// TwinCAT 3 PLC project Untitled1
// ProgramVersion: 3.1.4023.0
// libraries:
//   CmpBitmapPool, * (System)
//   Tc2_ControllerToolbox, * (Beckhoff Automation GmbH)
//   Tc2_Drive, * (Beckhoff Automation GmbH)
//   Tc2_EtherCAT, * (Beckhoff Automation GmbH)
//   Tc2_MC2, * (Beckhoff Automation GmbH)
//   Tc2_MC2_Camming, * (Beckhoff Automation GmbH)
//   Tc2_MC2_Drive, * (Beckhoff Automation GmbH)
//   Tc2_MC2_FlyingSaw, * (Beckhoff Automation GmbH)
//   Tc2_Standard, * (Beckhoff Automation GmbH)
//   Tc2_System, * (Beckhoff Automation GmbH)
//   Tc2_TcpIp, * (Beckhoff Automation GmbH)
//   Tc2_Utilities, * (Beckhoff Automation GmbH)
//   Tc3_Module, * (Beckhoff Automation GmbH)
//   VisuDialogs, * (System)
//   Visu Utils, * (System)
//   VisuSymbols,3.5.10.0,System
// project tree:
//   DUTs/Ctrl/ Cmd_Typ.TcDUT, Ctrl_Typ.TcDUT, InverterCtrl_Typ.TcDUT, Parameters_Typ.TcDUT, Persistent_Typ.TcDUT, Status_Typ.TcDUT, UnwindCmd_Typ.TcDUT, UnwinderParameters_Typ.TcDUT
//   DUTs/IO/Encoder/ Encoder_Control_Typ.TcDUT, Encoder_Status_Typ.TcDUT, Encoder_Typ.TcDUT
//   DUTs/IO/ IO_In_Typ.TcDUT, IO_Out_Typ.TcDUT, IO_Typ.TcDUT, ST_BasicInverter.TcDUT, ST_InfoData.TcDUT, ST_WcState.TcDUT
//   DUTs/Motion/Axis Typ/Basic Typ/ Basic_axis_typ.TcDUT
//   DUTs/Motion/Axis Typ/Basic Typ/enumTyp/ eBasicAxisState.TcDUT, eDriveModeOfOperation.TcDUT, eHomeModeOption.TcDUT, enumDriveType.TcDUT, enumMotionObject.TcDUT, enum_DriveUpdateError.TcDUT, enum_DriveUpdateStatus.TcDUT, E_EncoderType.TcDUT
//   DUTs/Motion/Axis Typ/Basic Typ/Input/ Basic_Input_typ.TcDUT
//   DUTs/Motion/Axis Typ/Basic Typ/Input/Cmd/ Basic_Command_axis_typ.TcDUT
//   DUTs/Motion/Axis Typ/Basic Typ/Input/Params/ Bacis_Parameter_axis_typ.TcDUT, Drive_Parameter_typ.TcDUT, Motion_Limit_Parameter.TcDUT, ST_BasicHomeParam.TcDUT, ST_HomeAbsEncoder.TcDUT, ST_HomeAbsSwitch.TcDUT, ST_HomeLagErr.TcDUT, ST_HomeOptions.TcDUT
//   DUTs/Motion/Axis Typ/Basic Typ/Output/ Basic_Error_axis_typ.TcDUT, Basic_Output_typ.TcDUT
//   DUTs/Motion/Axis Typ/Basic Typ/Output/Monitor/ Basic_Monitor_axis_typ.TcDUT, Basic_Monitor_FileUpdate_axis_typ.TcDUT
//   DUTs/Motion/Axis Typ/Basic Typ/Output/Status/ Basic_MC_MoveVelocity_Status_typ.TcDUT, Basic_MC_Power_Status_typ.TcDUT, Basic_MC_Reset_Status_typ.TcDUT, Basic_MC_SetOverride_typ.TcDUT, Basic_Status_axis_typ.TcDUT, Basic_Status_typ.TcDUT, Drive_Status_typ.TcDUT, ReadStatus_typ.TcDUT
//   DUTs/Motion/Axis Typ/CyclicAxis_Typ/ CyclicAxis_CMD_typ.TcDUT, CyclicAxis_Error_typ.TcDUT, CyclicAxis_Input_typ.TcDUT, CyclicAxis_monitor_typ.TcDUT, CyclicAxis_Output_typ.TcDUT, CyclicAxis_Param_typ.TcDUT, CyclicAxis_Status_typ.TcDUT, CyclicAxis_typ.TcDUT, CyclicPos_CMD_typ.TcDUT, CyclicPos_Param_typ.TcDUT, CyclicPos_Status_typ.TcDUT, CyclicVel_CMD_typ.TcDUT, CyclicVel_Param_typ.TcDUT, CyclicVel_Status_typ.TcDUT, eCyclicAxisState.TcDUT
//   DUTs/Motion/Axis Typ/ ExtendedAxisTyp_1.TcDUT, stAxisIF.TcDUT
//   DUTs/Motion/Axis Typ/MultiAxis_Typ/ CamIn_CMD_typ.TcDUT, CamIn_Param_typ.TcDUT, CamIn_Statuses_typ.TcDUT, CamOut_Param_typ.TcDUT, CamOut_Statuses_typ.TcDUT, CamTableSelectCMD_typ.TcDUT, CamTableSelect_Param_typ.TcDUT, CamTableSelect_Status_typ.TcDUT, eMultiAxisState.TcDUT, GearInDyn_CMD_typ.TcDUT, GearInDyn_Param_typ.TcDUT, GearInDyn_Statuses_typ.TcDUT, GearInMultiMaster_CMD_typ.TcDUT, GearInMultiMaster_Param_typ.TcDUT, GearInMultiMaster_Statuses_typ.TcDUT, GearInPos_CMD_typ.TcDUT, GearInPos_Param_typ.TcDUT, GearInPos_Statuses_typ.TcDUT, GearOut_Param_typ.TcDUT, GearOut_Statuses_typ.TcDUT, MultiAxis_CMD_typ.TcDUT, MultiAxis_Error_typ.TcDUT, MultiAxis_Input_typ.TcDUT, MultiAxis_monitor_typ.TcDUT, MultiAxis_Output_typ.TcDUT, MultiAxis_Param_typ.TcDUT, MultiAxis_Statuses_typ.TcDUT, MultiAxis_Status_typ.TcDUT, MultiAxis_typ.TcDUT
//   DUTs/Motion/Axis Typ/ParIDAccess_Typ/ eParIDAccessState.TcDUT, ParIDAccess_CMD_typ.TcDUT, ParIDAccess_Error_typ.TcDUT, ParIDAccess_Input_typ.TcDUT, ParIDAccess_monitor_typ.TcDUT, ParIDAccess_Output_typ.TcDUT, ParIDAccess_Param_typ.TcDUT, ParIDAccess_Par_ReadCoedSdo_typ.TcDUT, ParIDAccess_Par_WriteCoedSdo_typ.TcDUT, ParIDAccess_Status_axis_typ.TcDUT, ParIDAccess_Status_typ.TcDUT, ParIDAccess_Typ.TcDUT
//   DUTs/Motion/Axis Typ/VelocityCtrl/ eTorqueMode.TcDUT, eVelocityCtrlState.TcDUT, VelocityCtrl_CMD_typ.TcDUT, VelocityCtrl_Error_typ.TcDUT, VelocityCtrl_Input_typ.TcDUT, Velocityctrl_monitor_typ.TcDUT, VelocityCtrl_Output_typ.TcDUT, VelocityCtrl_Param_typ.TcDUT, VelocityCtrl_Status_typ.TcDUT, VelocityCtrl_typ.TcDUT
//   DUTs/Motion/ CoE_Obj_typ.TcDUT, ExtendedAxisTyp.TcDUT, STRUCT_AxisExtendedCompound.TcDUT, WebAxes_typ.TcDUT
//   DUTs/Motion/Enums/ eMotorID.TcDUT, eSensorID.TcDUT, eStationNo.TcDUT, eSubsystemID.TcDUT, eVendorNameID.TcDUT
//   DUTs/Motion/Winders/ DancerTyp.TcDUT, Dimeter_Typ.TcDUT, E_DancerCtrlTyp.TcDUT, Tension_Typ.TcDUT, WinderParam_Typ.TcDUT
//   / GlobalTextList.TcGTLO, VISU_TASK.TcTTO
//   GVLs/ AxesList.TcGVL, Consts.TcGVL, GVL.TcGVL, Persist.TcGVL
//   POUs/App/ FB_DancerCtrl.TcPOU, FB_HeaterProtection.TcPOU, FB_Machine_Ctrl.TcPOU, FB_Machine_Run.TcPOU, FB_Mechinit.TcPOU, FB_MechinitOutput.TcPOU, FB_OFF.TcPOU, FB_RW_Ctrl.TcPOU
//   POUs/Lib/CH Obj/CH_Typ/ Basic_cycle_CMD_typ.TcDUT, Basic_cycle_Input.TcDUT, Basic_cycle_Mon_typ.TcDUT, Basic_cycle_Output.TcDUT, Basic_cycle_Param_typ.TcDUT, Basic_cycle_Status_typ.TcDUT, Basic_cycle_typ.TcDUT, CH_ErrorReport_typ.TcDUT, Error_Handler_typ.TcDUT
//   POUs/Lib/CH Obj/ CycleHandleFB.TcPOU
//   POUs/Lib/Events/Demo/ DemoProgram.TcPOU
//   POUs/Lib/Events/Enums/ eMotorID_1.TcDUT, eSensorID_1.TcDUT, eStationNo_1.TcDUT, eSubsystemID_1.TcDUT, eVendorNameID_1.TcDUT
//   POUs/Lib/Events/ EventHelper.TcPOU, EventQueue.TcPOU
//   POUs/Lib/Events/Struct/ EventHeader_Typ.TcDUT, EventParam_Typ.TcDUT, EventReport_Typ.TcDUT
//   POUs/Lib/ FB_TensionLoop.TcPOU, Trigger.TcPOU
//   POUs/Lib/Inveter_Lib/ Enum_INV_Ctrl.TcDUT, Enum_INV_Status.TcDUT, FB_INV.TcPOU
//   POUs/Lib/IO/ fb_IO_Basic.TcPOU, fb_io_in_bool.TcPOU
//   POUs/Lib/Logging/HpString/ AMSNETID_TO_STRING.TcPOU, F_ADStoStr.TcPOU, itoax.TcPOU, strcmp.TcPOU, strcpy.TcPOU, strlen.TcPOU
//   POUs/Lib/Logging/logLib/DUTs/ enumLogMessageLevelSeverity.TcDUT, E_LogStatusReport_Type.TcDUT, FailureReportMsgStruct.TcDUT, LogArrayHandlePointers.TcDUT, LogArrayStruct.TcDUT, LogGlobalArrayObj.TcDUT, LogGlobalArraySemStruct.TcDUT, LogLocalArrayObj.TcDUT, LogMsgLogData.TcDUT, OperationTypeEnum.TcDUT
//   POUs/Lib/Logging/logLib/ fnLogMsg.TcPOU, fnLogMsg6.TcPOU, fnLogMsgInit.TcPOU, fnLogStatusToString.TcPOU, fnLogTransfer.TcPOU, fnSuppressBlank.TcPOU, GVL_1.TcGVL, LogMsg.TcPOU
//   POUs/Lib/Logging/PackData/ getUsint.TcPOU, putString.TcPOU, putUdint.TcPOU, putUint.TcPOU, putUsint.TcPOU
//   POUs/Lib/Logging/PLC_ClientComm/UDP_Comm/PcComm/ fbPcTransmit.TcPOU, PcComm.TcGVL, PcTransmit.TcPOU, RTC.TcPOU, UDPClientHandler_typ.TcDUT, UDPClientOutputStatus_typ.TcDUT
//   POUs/Lib/Motion/ BasicAxis_FB.TcPOU, CreateNCErrMsgDetails.TcPOU, CyclicAxis_FB.TcPOU, FC_NcErrorMsg.TcPOU, MultiAxis_FB.TcPOU, ParIDAccess_FB.TcPOU, VelocityCtrlAxis_FB.TcPOU
//   POUs/Lib/Motion/CanOpenAxis/BeckHoff/ BeckHoff8xxxAxis_FB.TcPOU, BeckHoffBasicAxis_FB.TcPOU, BeckHoffIntegratedAxis_FB.TcPOU, bk5xxxBasicAxis_FB.TcPOU, el7xxxBasicAxis_FB.TcPOU, ep7xxxBasicAxis_FB.TcPOU
//   POUs/Lib/Motion/CanOpenAxis/ CoEDrive_Ctrl_Adr_typ.TcDUT, CoE_BasicAxis_FB.TcPOU, CoE_FOE_Ctrl_typ.TcDUT, eCaOpDriveModeOfOperation.TcDUT, eHomingMethods.TcDUT, e_Homing_Contol_Word.TcDUT, e_Homing_Status_Word.TcDUT, Homing_CoE_Ctrl_Paramters_typ.TcDUT
//   POUs/Lib/Motion/CanOpenAxis/DriveParID/ eDS402DriveParID.TcDUT, eElmoDriveParID.TcDUT, eNidecDriveParID.TcDUT
//   POUs/Lib/Motion/CanOpenAxis/EcCoeSdo/ EcCoeSdo_Ctrl_typ.TcDUT, EcCoeSdo_Input_typ.TcDUT, EcCoeSdo_Output_typ.TcDUT, EcCoeSdo_Par_Read_typ.TcDUT, EcCoeSdo_Par_Write_typ.TcDUT, EcCoeSdo_Status_typ.TcDUT
//   POUs/Lib/Motion/CanOpenAxis/Elmo/ ElmoBasicAxis_FB.TcPOU, ElmoVelocityCtrlAxis_FB.TcPOU, FB_ElmoIOsHandle.TcPOU
//   POUs/Lib/Motion/CanOpenAxis/Lti/ LtiBasicAxis_FB.TcPOU
//   POUs/Lib/Motion/CanOpenAxis/Nidic/ NidicBasicAxis_FB.TcPOU, NidicIntegratedAxis_FB.TcPOU
//   POUs/Lib/Motion/CanOpenAxis/ServTronix/ ServoTronixBasicAxis_FB.TcPOU
//   POUs/Lib/Motion/CanOpenAxis/stepIM/ stepIMBasicAxis_FB.TcPOU
//   POUs/Lib/Motion/Engineering/ SrampHp.TcPOU
//   POUs/Lib/Motion/ErrorHandling_Lib/ Eh_ErrorEntry_typ.TcDUT, FB_ErrorHandler.TcPOU
//   POUs/Lib/Motion/EtherCAT/SDO_RW/ Tc2_EtherCAT_FB.TcPOU
//   POUs/Lib/Motion/EtherCAT/SDO_RW/Tc2_EtherCAT_typ/ EcCoeSdoRead_CMD_typ.TcDUT, EcCoeSdoRead_Param_typ.TcDUT, EcCoeSdoRead_Status_typ.TcDUT, EcCoeSdoWrite_CMD_typ.TcDUT, EcCoeSdoWrite_Param_typ.TcDUT, EcCoeSdoWrite_Status_typ.TcDUT, EcSoeRead_CMD_typ.TcDUT, EcSoeRead_Param_typ.TcDUT, EcSoeRead_Status_typ.TcDUT, EcSoeWrite_CMD_typ.TcDUT, EcSoeWrite_Param_typ.TcDUT, EcSoeWrite_Status_typ.TcDUT, Tc2_EtherCAT_Command_axis_typ.TcDUT, Tc2_EtherCAT_Error_typ.TcDUT, Tc2_EtherCAT_Input_typ.TcDUT, Tc2_EtherCAT_Output_typ.TcDUT, Tc2_EtherCAT_Parameter_axis_typ.TcDUT, Tc2_EtherCAT_Statuses_typ.TcDUT, Tc2_EtherCAT_typ.TcDUT
//   POUs/Lib/Motion/External Libs/Data types/ exCONSTANTS_MATH.TcDUT, exCONSTANTS_PHYS.TcDUT
//   POUs/Lib/Motion/External Libs/ exARRAY_MAX.TcPOU, exARRAY_MIN.TcPOU, exBIT_COUNT.TcPOU, exCHR_TO_STRING.TcPOU, exDWORD_TO_STRF.TcPOU, exD_TRUNC.TcPOU, exEVEN.TcPOU, exFILL.TcPOU, exFIX.TcPOU, exFRACT.TcPOU, exF_POWER.TcPOU, exINC1.TcPOU, exRDM.TcPOU, exRDM2.TcPOU, exTC_S.TcPOU, exTEMP_NTC.TcPOU, exTOGGLE.TcPOU, exT_PLC_MS.TcPOU, exT_PLC_US.TcPOU, ex_ARRAY_MEDIAN.TcPOU, ex_ARRAY_SORT.TcPOU, ex_ARRAY_SORT_LREAL.TcPOU, ex_ARRAY_SUM.TcPOU
//   POUs/Lib/Motion/External Libs/Global Variables/ exConstants.TcGVL, exGlobale_Variablen.TcGVL
//   POUs/Lib/Motion/FailureRport/Motor/ enumFailReportControlFailures.TcDUT, enumFailReportFailureType.TcDUT, enumFailReportMotorFailures.TcDUT, enumFailReportSeverity.TcDUT, enumMotorEvents.TcDUT, MotorFailureReport_FB.TcPOU
//   POUs/Lib/Motion/FailureRport/Terminal/Group/ TerminalGroupReport_FB.TcPOU, Terminal_Group_Ctrl_typ.TcDUT, Terminal_Group_Input_typ.TcDUT, Terminal_Group_Monitor_typ.TcDUT, Terminal_Group_Output_typ.TcDUT, Terminal_Group_Parameter_typ.TcDUT, Terminal_Group_Status_typ.TcDUT
//   POUs/Lib/Motion/FailureRport/Terminal/Terminal/ Terminal_Ctrl_typ.TcDUT, Terminal_Input_typ.TcDUT, Terminal_Monitor_typ.TcDUT, Terminal_Output_typ.TcDUT, Terminal_Parameter_typ.TcDUT, Terminal_Status_typ.TcDUT
//   POUs/Lib/Motion/SercosAxis/BeckHoff/ Beck5xxxAxis_FB.TcPOU
//   POUs/Lib/Motion/SercosAxis/ SercosBasicAxis_FB.TcPOU, SercosDrive_Ctrl_Adr_typ.TcDUT
//   POUs/Lib/ProgramBasic/ FB_PrgmBasic.TcPOU, LocalEvent_Typ.TcDUT
//   POUs/Lib/Signal/ E_LutMode.TcDUT, FB_LPF.TcPOU, LookUP_Table.TcPOU, ST_LookUpTableParam.TcDUT
//   POUs/Lib/System/CmdQueue/DUTs/ DelayInfo_typ.TcDUT, eDelayType.TcTLEO
//   POUs/Lib/System/CmdQueue/ FB_CmdQueue.TcPOU
//   POUs/Lib/System/ fAnalogSensorScale.TcPOU, FB_BaseFb.TcPOU, FB_FileEntireReadAtomic.TcPOU, fnCnvToTarg.TcPOU, Queue.TcPOU
//   POUs/ MAIN.TcPOU, prg_Motion.TcPOU
//   TasksRef/ PlcTask.TcTTO, Task2ms.TcTTO
//   VISUs/Dialogs/ DialogTimer.TcVIS, DialogTimer_ColdCut.TcVIS, DialogTimer_GripperPosi.TcVIS, DialogTimer_HeaterOff.TcVIS, DialogTimer_GripperOpenClose.TcVIS, DialogTimer_HotWeldValve.TcVIS, DialogTimer_HeaterOn.TcVIS, DialogTimer_ValveClose.TcVIS, Dialog_Estop.TcVIS, Dialog_IO.TcVIS, Dialog_Output.TcVIS, Dialog_Settings.TcVIS, Winders.TcVIS
//   VISUs/ HMI.TcPOU, ImagePool.TcIPO (not stored), Visualization.TcVIS, VisualizationManager.TcVMO (not stored)
//   VISUs/Img/ MachineState.TcTLO
//   VISUs/infra/ CloseDialog.TcPOU, OpenDialog.TcPOU
// real-time tasks:
//   TASK PlcTask: cycle T#10ms, priority 20, ADS port 350
//   TASK VISU_TASK: cycle T#200000us, priority 30, ADS port 351
//   TASK Task2ms: cycle T#2ms, priority 1, ADS port 352
// motion (NC):
//   TASK NC-Task 1 SAF: cycle T#2ms, priority 4, ADS port 501
//   TASK NC-Task 1 SVB: cycle T#2ms, priority 8, ADS port 511
//   AXIS UW_1 (id 11)
//     General: IoDivider=3
//     Dynamic: AccelerationMaximum=30000000, DecelerationMaximum=30000000, Acceleration=3336590, Deceleration=3336590, Jerk=10009800
//     Velo: RefSearch=22243.9024390244, RefSync=22243.9024390244, SlowManual=200000, FastManual=500000, Fast=2224390.24390244, Maximum=2224390
//     PositionAreaControl: Enable=false
//     TargetPosControl: Enable=false
//     OtherSettings: ErrorReactionMode=1, ErrorReactionDelay=5, AllowMotionCmdToSlave=true
//     encoder EncType=8
//       EncPara: ScaleFactorNumerator=35121.9512195122, ScaleFactorDenominator=1048576, Inverse=true, MaxCount=#xffffffff
//     drive DrvType=9
//       DrvPara: Inverse=true, MaxCount=#xffffffff, DriveControlDWord=#x00000100
//         Analog: VeloReferenz=2446829.26829268, VeloScale=1.02400649589962, TorqueSetpointScale=10, ScaleFactorActTorque=0.1
//         TimeComp: TaskDelayCycles=1
//     controller CtrType=1
//       CtrPara: PriorControlFactor=1
//         PosDiffControl: Enable=false
//         PID: PosKp=10
//         Observer: BandWidth=20
//   AXIS UW_V_master (id 31)
//     General: IoDivider=3
//     Dynamic: AccelerationMaximum=30000000, DecelerationMaximum=30000000, Acceleration=1000000, Deceleration=1000000, Jerk=300000000
//     Velo: Maximum=3000000
//     OtherSettings: ErrorReactionMode=1, ErrorReactionDelay=5, AllowMotionCmdToSlave=true
//     encoder EncType=1
//     drive DrvType=5
//       Analog: VeloReferenz=3000000, ScaleFactorActTorque=0.1
//       TimeComp: TaskDelayCycles=1
//     controller CtrType=1
//       CtrPara: PriorControlFactor=1
//         Observer: BandWidth=20
//   AXIS UW_2 (id 1)
//     General: IoDivider=3
//     Dynamic: AccelerationMaximum=30000000, DecelerationMaximum=30000000, Acceleration=3336590, Deceleration=3336590, Jerk=10009800
//     Velo: RefSearch=22243.9024390244, RefSync=22243.9024390244, SlowManual=200000, FastManual=500000, Fast=2224390.24390244, Maximum=2224390
//     PositionAreaControl: Enable=false
//     TargetPosControl: Enable=false
//     OtherSettings: ErrorReactionMode=1, ErrorReactionDelay=5, AllowMotionCmdToSlave=true
//     encoder EncType=8
//       EncPara: ScaleFactorNumerator=35121.9512195122, ScaleFactorDenominator=1048576, Inverse=true, MaxCount=#xffffffff
//     drive DrvType=9
//       DrvPara: Inverse=true, MaxCount=#xffffffff, DriveControlDWord=#x00000100
//         Analog: VeloReferenz=2446829.26829268, VeloScale=1.02400649589962, TorqueSetpointScale=10, ScaleFactorActTorque=0.1
//         TimeComp: TaskDelayCycles=1
//     controller CtrType=1
//       CtrPara: PriorControlFactor=1
//         PosDiffControl: Enable=false
//         PID: PosKp=0
//         Observer: BandWidth=20
//   AXIS OutAxis (id 2)
//     Dynamic: Acceleration=15000, Deceleration=15000, Jerk=15000
//     Velo: Maximum=5000
//     PositionAreaControl: Enable=false
//     TargetPosControl: Enable=false
//     OtherSettings: AllowMotionCmdToSlave=true
//     encoder EncType=19
//       EncPara: ScaleFactorNumerator=75, ScaleFactorDenominator=8192, MaxCount=#xffffffff
//     drive DrvType=16
//       DrvPara: MaxCount=#xffffffff, DriveControlDWord=#x00020000
//         Analog: VeloReferenz=5000, VeloScale=125, TorqueSetpointScale=10, ScaleFactorActTorque=0.1
//         TimeComp: TaskDelayCycles=1
//     controller CtrType=1
//       CtrPara: PriorControlFactor=1
//         PosDiffControl: Enable=false
//         PID: PosKp=0
//         Observer: BandWidth=20
// I/O:
//   DEVICE Device 1 (EtherCAT), AmsNetId 192.168.101.10.2.1
//     Term 1 (EK1100) [EK1100 EtherCAT Coupler (2A E-Bus)]
//       Term 2 (EL4004) [EL4004 4Ch. Ana. Output 0-10V, 12bit]
//       Term 3 (EL1859) [EL1859 8Ch. Dig. Input 24V, 3ms, 8Ch. Dig. Output 24V, 0.5A]
//       Term 4 (EL1859) [EL1859 8Ch. Dig. Input 24V, 3ms, 8Ch. Dig. Output 24V, 0.5A]
//       Term 5 (EL3004) [EL3004 4Ch. Ana. Input +/-10V]
//       Term 6 (EL3054) [EL3054 4Ch. Ana. Input 4-20mA]
//       Term 7 (EL9510) [EL9510 Power supply terminal 10V]
//       UW2_loadCell_ (EL3356-0010) [EL3356-0010 1Ch. Ana. Input Resistor Bridge Terminal, 24bit, High Precision]
//       UW1_loadCel (EL3356-0010) [EL3356-0010 1Ch. Ana. Input Resistor Bridge Terminal, 24bit, High Precision]
//       Term 7 (EL6070-1208) [EL6070-1208 1Ch. Licensing-Terminal]
//       Term 28 (EL9011) [EL9011 End Terminal]
//     UW_1_Axis (AX5106-0000-0203) [AX5106-0000-0203 EtherCAT Drive (SoE, 1 Ch.)]
//     Drive 1 (AX5106-0000-0203) [AX5106-0000-0203 EtherCAT Drive (SoE, 1 Ch.)]
//     Drive 27 (Elmo Drive ) [Gold EtherCAT GCON Drive ID Selector Rev:0x00010420]
// variable links:
//   NC-Task 1 SAF/Axes/OutAxis <-> Device 1 (EtherCAT)/Drive 27 (Elmo Drive )
//     Drive/Inputs/In/nDcOutputTime <-> InfoData/DcOutputShift
//     Drive/Inputs/In/nState1 <-> Inputs/Status word
//     Drive/Inputs/In/nState2 <-> Inputs/Status word @bit 8
//     Drive/Inputs/In/nState4 @bit 1 <-> WcState/InputToggle
//     Drive/Inputs/In/nState4 <-> WcState/WcState
//     Drive/Outputs/Out/nCtrl1 <-> Outputs/Control word
//     Drive/Outputs/Out/nCtrl2 <-> Outputs/Control word @bit 8
//     Drive/Outputs/Out/nDataOut1 <-> Outputs/Target Position
//     Drive/Outputs/Out/nDataOut2 <-> Outputs_1/Velocity Offset
//     Enc/Inputs/In/nDataIn1 <-> Inputs/Position actual value
//     Enc/Inputs/In/nDcInputTime <-> InfoData/DcInputShift
//     Enc/Inputs/In/nState4 @bit 1 <-> WcState/InputToggle
//     Enc/Inputs/In/nState4 <-> WcState/WcState
//   Untitled1/Untitled1 Instance <-> Device 1 (EtherCAT)/Term 1 (EK1100)/Term 3 (EL1859)
//     PlcTask Inputs/GVL.gMachineCtrl.IO.In.E_StopPressedRaw <-> Channel 1/GVL.gMachineCtrl.IO.In.E_StopPressedRaw
//     PlcTask Outputs/GVL.gMachineCtrl.IO.Out.Buzzer <-> Channel 15/Output
//     PlcTask Outputs/GVL.gMachineCtrl.IO.Out.ExternalNipMotor <-> Channel 14/Output
//     PlcTask Outputs/GVL.gMachineCtrl.IO.Out.Output_GripperClose <-> Channel 12/Output
//     PlcTask Outputs/GVL.gMachineCtrl.IO.Out.Output_GripperOpen <-> Channel 13/Output
//   Untitled1/Untitled1 Instance <-> Device 1 (EtherCAT)/Term 1 (EK1100)/Term 4 (EL1859)
//     PlcTask Inputs/GVL.gMachineCtrl.IO.In.GripperEndPosition <-> Channel 8/Input
//     PlcTask Inputs/GVL.gMachineCtrl.IO.In.GripperStartPosition <-> Channel 7/Input
//     PlcTask Inputs/GVL.gMachineCtrl.IO.In.HomeOutAxis <-> Channel 3/Input
//     PlcTask Inputs/GVL.gMachineCtrl.IO.In.HomeOutAxisLimit <-> Channel 4/Input
//     PlcTask Inputs/GVL.gMachineCtrl.IO.In.UW_1_DancerEmpetyRaw <-> Channel 5/Input
//     PlcTask Inputs/GVL.gMachineCtrl.IO.In.UW_2_DancerEmpetyRaw <-> Channel 6/Input
//     PlcTask Inputs/GVL.gMachineCtrl.IO.In.UW_1_DancerFullRaw <-> Channel 1/Input
//     PlcTask Inputs/GVL.gMachineCtrl.IO.In.UW_2_DancerFullRaw <-> Channel 2/Input
//     PlcTask Outputs/GVL.gMachineCtrl.IO.Out.ColdCutPistonDown <-> Channel 10/Output
//     PlcTask Outputs/GVL.gMachineCtrl.IO.Out.GripperOpen <-> Channel 13/Output
//     PlcTask Outputs/GVL.gMachineCtrl.IO.Out.GripperPistonPosition <-> Channel 14/Output
//     PlcTask Outputs/GVL.gMachineCtrl.IO.Out.GripperRetract <-> Channel 12/Output
//     PlcTask Outputs/GVL.gMachineCtrl.IO.Out.HeaterOn <-> Channel 15/Output
//     PlcTask Outputs/GVL.gMachineCtrl.IO.Out.KniveCut <-> Channel 11/Output
//     PlcTask Outputs/GVL.gMachineCtrl.IO.Out.PressDown <-> Channel 9/Output
//   Untitled1/Untitled1 Instance <-> Device 1 (EtherCAT)/Term 1 (EK1100)/Term 5 (EL3004)
//     Task2ms Inputs/GVL.gMachineCtrl.IO.In.UW_1_Diameter <-> AI Standard Channel 2/Value
//     Task2ms Inputs/GVL.gMachineCtrl.IO.In.UW_2_Diameter <-> AI Standard Channel 1/Value
//   Untitled1/Untitled1 Instance <-> Device 1 (EtherCAT)/Term 1 (EK1100)/UW1_loadCel (EL3356-0010)
//     Task2ms Inputs/GVL.gMachineCtrl.IO.In.UW_1_LoacCell <-> RMB Value (INT32)/Value
//   Untitled1/Untitled1 Instance <-> Device 1 (EtherCAT)/Term 1 (EK1100)/UW2_loadCell_ (EL3356-0010)
//     Task2ms Inputs/GVL.gMachineCtrl.IO.In.UW_2_LoacCell <-> RMB Value (INT32)/Value
//   Untitled1/Untitled1 Instance <-> Device 1 (EtherCAT)/UW_1_Axis (AX5106-0000-0203)
//     PlcTask Inputs/MAIN.uw1_Toque <-> AT/Torque feedback value
//   Untitled1/Untitled1 Instance <-> NC-Task 1 SAF/Axes/OutAxis
//     Task2ms Inputs/AxesList.gWebAxes.Output.Ref.NcToPlc <-> Outputs/ToPlc
//     Task2ms Outputs/AxesList.gWebAxes.Output.Ref.PlcToNc <-> Inputs/FromPlc
//   Untitled1/Untitled1 Instance <-> NC-Task 1 SAF/Axes/UW_1
//     Task2ms Inputs/AxesList.gWebAxes.UW_1.Ref.NcToPlc <-> Outputs/ToPlc
//     Task2ms Outputs/AxesList.gWebAxes.UW_1.Ref.PlcToNc <-> Inputs/FromPlc
//   Untitled1/Untitled1 Instance <-> NC-Task 1 SAF/Axes/UW_2
//     Task2ms Inputs/AxesList.gWebAxes.UW_2.Ref.NcToPlc <-> Outputs/ToPlc
//     Task2ms Outputs/AxesList.gWebAxes.UW_2.Ref.PlcToNc <-> Inputs/FromPlc
//   Untitled1/Untitled1 Instance <-> NC-Task 1 SAF/Axes/UW_V_master
//     Task2ms Inputs/AxesList.gWebAxes.UwVmaster.Ref.NcToPlc <-> Outputs/ToPlc
//     Task2ms Outputs/AxesList.gWebAxes.UwVmaster.Ref.PlcToNc <-> Inputs/FromPlc
//   __THIS__ <-> Device 1 (EtherCAT)/UW_1_DRV (AX5106-0000-0213)
//     Drive/Inputs/In/nDataIn1 <-> AT/Following distance
//     Drive/Inputs/In/nDataIn3[0] <-> AT/Torque/force feedback value
//     Drive/Inputs/In/nDcOutputTime <-> InfoData/DcOutputShift
//     Drive/Inputs/In/nState1 <-> AT/Drive status word @bit 8
//     Drive/Inputs/In/nState2 <-> AT/Drive status word
//     Drive/Inputs/In/nState4 @bit 1 <-> WcState/InputToggle
//     Drive/Inputs/In/nState4 <-> WcState/WcState
//     Drive/Outputs/Out/nCtrl1 <-> MDT/Master control word @bit 8
//     Drive/Outputs/Out/nDataOut1 <-> MDT/Position command value
//     Enc/Inputs/In/nDataIn1 <-> AT/Position feedback 1 value
//     Enc/Inputs/In/nDcInputTime <-> InfoData/DcInputShift
//     Enc/Inputs/In/nState4 @bit 1 <-> WcState/InputToggle
//     Enc/Inputs/In/nState4 <-> WcState/WcState
//   __THIS__ <-> Untitled1/Untitled1 Instance
//     Inputs/FromPlc <-> PlcTask Outputs/AxesList.gWebAxes.UW_1.Ref.PlcToNc
//     Outputs/ToPlc <-> PlcTask Inputs/AxesList.gWebAxes.UW_1.Ref.NcToPlc
//     Inputs/FromPlc <-> Task2ms Outputs/AxesList.gWebAxes.UW_1.Ref.PlcToNc
//     Inputs/FromPlc <-> Task2ms Outputs/AxesList.gWebAxes.UW_2.Ref.PlcToNc
//     Outputs/ToPlc <-> Task2ms Inputs/AxesList.gWebAxes.UW_1.Ref.NcToPlc
//     Outputs/ToPlc <-> Task2ms Inputs/AxesList.gWebAxes.UW_2.Ref.NcToPlc
//     Inputs/FromPlc <-> PlcTask Outputs/AxesList.gWebAxes.UwVmaster.Ref.PlcToNc
//     Outputs/ToPlc <-> PlcTask Inputs/AxesList.gWebAxes.UwVmaster.Ref.NcToPlc
//     Inputs/FromPlc <-> Task2ms Outputs/AxesList.gWebAxes.UwVmaster.Ref.PlcToNc
//     Outputs/ToPlc <-> Task2ms Inputs/AxesList.gWebAxes.UwVmaster.Ref.NcToPlc
//   __THIS__ <-> Device 1 (EtherCAT)/UW_1_Axis (AX5106-0000-0203)
//     Drive/Inputs/In/nDataIn1 <-> AT/Following distance
//     Drive/Inputs/In/nDataIn3[0] <-> AT/Torque feedback value
//     Drive/Inputs/In/nDcOutputTime <-> InfoData/DcOutputShift
//     Drive/Inputs/In/nState1 <-> AT/Drive status word @bit 8
//     Drive/Inputs/In/nState2 <-> AT/Drive status word
//     Drive/Inputs/In/nState4 @bit 1 <-> WcState/InputToggle
//     Drive/Inputs/In/nState4 <-> WcState/WcState
//     Drive/Outputs/Out/nCtrl1 <-> MDT/Master control word @bit 8
//     Drive/Outputs/Out/nDataOut1 <-> MDT/Position command value
//     Enc/Inputs/In/nDataIn1 <-> AT/Position feedback 1 value
//     Enc/Inputs/In/nDcInputTime <-> InfoData/DcInputShift
//     Enc/Inputs/In/nState4 @bit 1 <-> WcState/InputToggle
//     Enc/Inputs/In/nState4 <-> WcState/WcState
//   (this object) <-> Device 1 (EtherCAT)/UW_1_Axis (AX5106-0000-0203)
//     Drive/Inputs/In/nDataIn1 <-> AT/Following distance
//     Drive/Inputs/In/nDataIn3[0] <-> AT/Torque feedback value
//     Drive/Inputs/In/nDcOutputTime <-> InfoData/DcOutputShift
//     Drive/Inputs/In/nState1 <-> AT/Drive status word @bit 8
//     Drive/Inputs/In/nState2 <-> AT/Drive status word
//     Drive/Inputs/In/nState4 @bit 1 <-> WcState/InputToggle
//     Drive/Inputs/In/nState4 <-> WcState/WcState
//     Drive/Outputs/Out/nCtrl1 <-> MDT/Master control word @bit 8
//     Drive/Outputs/Out/nDataOut1 <-> MDT/Position command value
//     Enc/Inputs/In/nDataIn1 <-> AT/Position feedback 1 value
//     Enc/Inputs/In/nDcInputTime <-> InfoData/DcInputShift
//     Enc/Inputs/In/nState4 @bit 1 <-> WcState/InputToggle
//     Enc/Inputs/In/nState4 <-> WcState/WcState
//   __THIS__ <-> OCB/OCB Instance
//     Inputs/FromPlc <-> Task_C1_008ms Outputs/AxesList.gWebAxes.UwVmaster.Ref.PlcToNc
//     Outputs/ToPlc <-> Task_C1_008ms Inputs/AxesList.gWebAxes.UwVmaster.Ref.NcToPlc
//   __THIS__ <-> Device 1 (EtherCAT)/Drive 1 (AX5106-0000-0203)
//     Drive/Inputs/In/nDataIn1 <-> AT/Following distance
//     Drive/Inputs/In/nDcOutputTime <-> InfoData/DcOutputShift
//     Drive/Inputs/In/nState1 <-> AT/Drive status word @bit 8
//     Drive/Inputs/In/nState2 <-> AT/Drive status word
//     Drive/Inputs/In/nState4 @bit 1 <-> WcState/InputToggle
//     Drive/Inputs/In/nState4 <-> WcState/WcState
//     Drive/Outputs/Out/nCtrl1 <-> MDT/Master control word @bit 8
//     Drive/Outputs/Out/nDataOut1 <-> MDT/Position command value
//     Enc/Inputs/In/nDataIn1 <-> AT/Position feedback 1 value
//     Enc/Inputs/In/nDcInputTime <-> InfoData/DcInputShift
//     Enc/Inputs/In/nState4 @bit 1 <-> WcState/InputToggle
//     Enc/Inputs/In/nState4 <-> WcState/WcState
//   (this object) <-> Device 1 (EtherCAT)/Drive 1 (AX5106-0000-0203)
//     Drive/Inputs/In/nDataIn1 <-> AT/Following distance
//     Drive/Inputs/In/nDcOutputTime <-> InfoData/DcOutputShift
//     Drive/Inputs/In/nState1 <-> AT/Drive status word @bit 8
//     Drive/Inputs/In/nState2 <-> AT/Drive status word
//     Drive/Inputs/In/nState4 @bit 1 <-> WcState/InputToggle
//     Drive/Inputs/In/nState4 <-> WcState/WcState
//     Drive/Outputs/Out/nCtrl1 <-> MDT/Master control word @bit 8
//     Drive/Outputs/Out/nDataOut1 <-> MDT/Position command value
//     Enc/Inputs/In/nDataIn1 <-> AT/Position feedback 1 value
//     Enc/Inputs/In/nDcInputTime <-> InfoData/DcInputShift
//     Enc/Inputs/In/nState4 @bit 1 <-> WcState/InputToggle
//     Enc/Inputs/In/nState4 <-> WcState/WcState

CONFIGURATION Untitled1
    RESOURCE PLC ON TwinCAT3
        TASK PlcTask(INTERVAL := T#10ms, PRIORITY := 20);
        TASK Task2ms(INTERVAL := T#2ms, PRIORITY := 1);
        TASK VISU_TASK(INTERVAL := T#200000us, PRIORITY := 30);
        PROGRAM MAIN WITH PlcTask : MAIN;
        PROGRAM prg_Motion WITH Task2ms : prg_Motion;
        PROGRAM VisuElems_Visu_Prg WITH VISU_TASK : VisuElems.Visu_Prg;
        PROGRAM HMI WITH VISU_TASK : HMI;
    END_RESOURCE
END_CONFIGURATION

// ---- DUTs/Ctrl/Cmd_Typ.TcDUT
TYPE Cmd_Typ :
STRUCT
	Start:BOOL;
	SwitchOn:BOOL;
	Manual:BOOL;
	Stop:BOOL;
	EmStop:BOOL;
	
	UW_1_Cmd : UnwindCmd_Typ;
	UW_2_Cmd : UnwindCmd_Typ;

	
END_STRUCT
END_TYPE

// ---- DUTs/Ctrl/Ctrl_Typ.TcDUT
TYPE Ctrl_Typ :
STRUCT
	Cmd:Cmd_Typ;
	RwInverter:InverterCtrl_Typ;
	Parameters:Parameters_Typ;
	IO:IO_Typ;
	Status:Status_Typ;
	
	Simulation:BOOL;
	Manual:BOOL;
END_STRUCT
END_TYPE

// ---- DUTs/Ctrl/InverterCtrl_Typ.TcDUT
TYPE InverterCtrl_Typ :
STRUCT
	Start:BOOL;
	ResetError:BOOL;
	SetVelocity:INT;
	ActualVelocity:INT;
END_STRUCT
END_TYPE

// ---- DUTs/Ctrl/Parameters_Typ.TcDUT
TYPE Parameters_Typ :
STRUCT
	//TimerPressDown1:DINT;//[MS]
	
	Continues:BOOL;
	NumberOfCycles:UDINT;
	WebLinarSpeed:LREAL;//[mm]
	WebLinarSpeedSlow:LREAL;//[mm]
	
	DancerFillSpeed :LREAL;//[Degrees per seconds]
	
	
	
	MotorVelocity :INT;
	DistanceToMove:UINT;
	
	
	OutGripperEndPosition:LREAL;
	OutGripperHomeVelocity:LREAL;
	OutGripperProcessVelocity:LREAL;
	
	
	UW_1_Param	: UnwinderParameters_Typ;
	UW_2_Param	: UnwinderParameters_Typ;
	
END_STRUCT
END_TYPE

// ---- DUTs/Ctrl/Persistent_Typ.TcDUT
TYPE Persistent_Typ :
STRUCT
	LifeTimerCounter:UDINT;
	//Timers
	TimeColdCutPressDown: DINT := 500;
	TimeGripperStartPosition: DINT := 20000;
	TimeGripperHomePosition: DINT := 7000;
	//TimeGripperMoveDelay: DINT := 3500;
	TimeGripperOpen: DINT := 3000;
	TimeOutputGripperClose: DINT := 3000;
	TimeGripperRetract: DINT := 4000;
	TimeHotWeldPressDown: DINT := 5000;
	TimerHotWeldingOn: DINT := 6000;
	TimerHotWeldingOff: DINT := 2000;
	TimerPressUp: DINT := 4000;
	
	TimeKniveVut: DINT := 3000;
	
	TimerMotorOn: DINT := 3000;
END_STRUCT
END_TYPE

// ---- DUTs/Ctrl/Status_Typ.TcDUT
TYPE Status_Typ :
STRUCT
	SessionCounter:UINT;
	UW_1_DancerFull:BOOL;
	UW_2_DancerFull:BOOL;
END_STRUCT
END_TYPE

// ---- DUTs/Ctrl/UnwindCmd_Typ.TcDUT
TYPE UnwindCmd_Typ :
STRUCT
	JogFwd:BOOL;
	JogBack:BOOL;
	JogSFwdSlow:BOOL;
	JogBackdSlow:BOOL;
	JogDancerFill:BOOL;	
END_STRUCT
END_TYPE

// ---- DUTs/Ctrl/UnwinderParameters_Typ.TcDUT
TYPE UnwinderParameters_Typ :
STRUCT
	ForceDiameter:BOOL;
	ForcedDiameter:LREAL;
	
	EnableTension:BOOL;
	SetTension:REAL;
	
	kp:LREAL;
	TN:TIME;
	
	kpMove:LREAL;
	TNMove:TIME;
	
	EnableDancer:BOOL;
	
END_STRUCT
END_TYPE

// ---- DUTs/IO/Encoder/Encoder_Control_Typ.TcDUT
TYPE Encoder_Control_Typ :
STRUCT
	SetCounterCmd AT %Q* 	: BOOL;
	SetCounterValue AT %Q* 	: UINT;
END_STRUCT
END_TYPE

// ---- DUTs/IO/Encoder/Encoder_Status_Typ.TcDUT
TYPE Encoder_Status_Typ :
STRUCT
	CounterValue AT %I* 	: UINT;
	SetCounterDone AT %I* 	: BOOL;
	
END_STRUCT
END_TYPE

// ---- DUTs/IO/Encoder/Encoder_Typ.TcDUT
TYPE Encoder_Typ :
STRUCT
	Status :Encoder_Status_Typ;
	Ctrl:Encoder_Control_Typ;
END_STRUCT
END_TYPE

// ---- DUTs/IO/IO_In_Typ.TcDUT
TYPE IO_In_Typ :
STRUCT
	PrimeryPressFeedback :fb_io_in_bool;
	SeconderyPressFeedbak:fb_io_in_bool;
	E_StopPressed  	: BOOL;
	E_StopPressedRaw AT %I* 	: BOOL;
	
	UW_1_Diameter AT %I* 	: INT;
	UW_2_Diameter AT %I* 	: INT;
	UW_1_LoacCell AT %I* 	: DINT;
	UW_2_LoacCell AT %I* 	: DINT;	
	
	UW_1_DancerFull  	: BOOL;
	UW_2_DancerFull  	: BOOL;
	
	UW_1_DancerFullRaw AT %I* 	: BOOL;
	UW_2_DancerFullRaw AT %I* 	: BOOL;	
	
	UW_1_DancerPosition AT %I* 	: INT;
	UW_2_DancerPosition AT %I* 	: INT;

	HomeOutAxis	 AT %I* 	: BOOL;
	HomeOutAxisLimit	 AT %I* 	: BOOL;
	
	GripperStartPosition	 AT %I* 	: BOOL;
	GripperEndPosition	 AT %I* 	: BOOL;
	
	UW_1_DancerEmpetyRaw AT %I* 	: BOOL;
	UW_2_DancerEmpetyRaw AT %I* 	: BOOL;
	
	UW_1_DancerEmpety AT %I* 	: BOOL;
	UW_2_DancerEmpety AT %I* 	: BOOL;	
	
END_STRUCT
END_TYPE

// ---- DUTs/IO/IO_Out_Typ.TcDUT
TYPE IO_Out_Typ :
STRUCT
	HeaterOn  		 			AT %Q* 	: BOOL;
	GripperOpen 	 			AT %Q* 	: BOOL;
	Output_GripperClose 	 			AT %Q* 	: BOOL;
	Output_GripperOpen 	 			AT %Q* 	: BOOL;
	GripperRetract 	 			AT %Q* 	: BOOL;
	GripperPistonPosition 		AT %Q* 	: BOOL;
	PressDown			 	 AT %Q* 	: BOOL;
	ColdCutPistonDown			 	 AT %Q* 	: BOOL;
	KniveCut			 	 AT %Q* 	: BOOL;
	
	ExternalNipMotor			 	 AT %Q* 	: BOOL;
	
	Buzzer			 	 AT %Q* 	: BOOL;
END_STRUCT
END_TYPE

// ---- DUTs/IO/IO_Typ.TcDUT
TYPE IO_Typ :
STRUCT
	In:IO_In_Typ;
	Out:IO_Out_Typ;
	EncoderRW:Encoder_Typ;
	//RwInverter:ST_BasicInverter;
END_STRUCT
END_TYPE

// ---- DUTs/IO/ST_BasicInverter.TcDUT
TYPE ST_BasicInverter :	
STRUCT
	StatusWord		AT %I* 	: UINT;
	ActualSpeed		AT %I*	: INT;
	ControlWord 	AT %Q* 	: UINT;
	SetSpeed		AT %Q*	: INT;
	InfoData				: ST_InfoData;
	stWcState 		AT %I*  : ST_WcState;	
END_STRUCT
END_TYPE

// ---- DUTs/IO/ST_InfoData.TcDUT
TYPE ST_InfoData :
STRUCT
	State  AT %I*	:	UINT;
	AdsAdr AT %I*	: 	AMSADDR;
END_STRUCT
END_TYPE

// ---- DUTs/IO/ST_WcState.TcDUT
TYPE ST_WcState :
STRUCT
	WcState		: BIT;
	InputToggle	: BIT;
END_STRUCT
END_TYPE

// ---- DUTs/Motion/Axis Typ/Basic Typ/Basic_axis_typ.TcDUT
TYPE Basic_axis_typ : 	
	STRUCT 
		Input : Basic_Input_typ; (*command structure*)
		Output : Basic_Output_typ; (*parameter structure*)
	END_STRUCT
END_TYPE

// ---- DUTs/Motion/Axis Typ/Basic Typ/enumTyp/eBasicAxisState.TcDUT
TYPE eBasicAxisState :
(
	BASIC_STATE_INIT := 0,
	BASIC_STATE_WAIT,
	BASIC_STATE_POWER_ON,
	BASIC_STATE_READY,
	BASIC_STATE_HOME,
	BASIC_STATE_STOP,
	BASIC_STATE_HALT,
	BASIC_STATE_MOVE_ABSOLUTE,
	BASIC_STATE_MOVE_ADDITIVE,
	BASIC_STATE_MOVE_RELATIVE,
	BASIC_STATE_MOVE_VELOCITY,
	BASIC_STATE_JOG_POSITIVE,
	BASIC_STATE_JOG_NEGATIVE,
	//BASIC_STATE_SET_OVERRIDE,
	BASIC_STATE_ERROR_RESET,
	BASIC_STATE_ERROR_AXIS,
	BASIC_STATE_ERROR,
	ENTER_ETHERCAT_FAILURE, 
	BASIC_STATE_NOT_ACTIVE
);
END_TYPE

// ---- DUTs/Motion/Axis Typ/Basic Typ/enumTyp/eDriveModeOfOperation.TcDUT
{attribute 'qualified_only'}
{attribute 'strict'}
TYPE eDriveModeOfOperation :
(
	ProfilePositionMode				:= 1,
	VelocityCtrMode    				:= 2,
	ProfileVelocityMode 	   	    := 3,
	TorqueVelocityMode 				:= 4,
	HomingMode				    	:= 6,
	InterpolationPosMode			:= 7,
	CyclicSyncMode					:= 8,
	CyclicSyncVelocity				:= 9,
	CyclicSyncTorque				:= 10
	
	
);
END_TYPE

// ---- DUTs/Motion/Axis Typ/Basic Typ/enumTyp/eHomeModeOption.TcDUT

TYPE eHomeModeOption :
(
	eNEGATIVE := 0 ,
	ePOSITIVE := 1
);
END_TYPE

// ---- DUTs/Motion/Axis Typ/Basic Typ/enumTyp/enumDriveType.TcDUT
{attribute 'qualified_only'}
{attribute 'strict'}
TYPE enumDriveType :
(
	eNoDrive := 0,
	eEL70xx,
	eEP70xx,
	eEL70xxExternFeedBack,
	eElmo,
	stepIM,
	eNidec,
	eIntegratedNidec,
	eIntegratedBeckhoff,
	e8xxxBeckhoff,
	e5xxxBeckhoff
);
END_TYPE

// ---- DUTs/Motion/Axis Typ/Basic Typ/enumTyp/enumMotionObject.TcDUT
{attribute 'qualified_only'}
{attribute 'strict'}
TYPE enumMotionObject :
(
	OPERATION_MODE := 1,	
	VEL_KI,
	VEL_KP,
	TORQUE_OFFSET,
	MAX_TORQUE,
	GAIN_SCHEDULE,
	ACC_CLOSE_POS_ERR,
	DC_VOLATAGE
	
	
);
END_TYPE

// ---- DUTs/Motion/Axis Typ/Basic Typ/enumTyp/enum_DriveUpdateError.TcDUT
{attribute 'qualified_only'}
{attribute 'strict'}
TYPE enum_DriveUpdateError :
(
	NoError,
	FileNotFound,
	FileClosedFailed,
	FoeFailed
);
END_TYPE

// ---- DUTs/Motion/Axis Typ/Basic Typ/enumTyp/enum_DriveUpdateStatus.TcDUT
{attribute 'qualified_only'}
{attribute 'strict'}
TYPE enum_DriveUpdateStatus :
(
	NoAction:= 0,
	Checking,
	UpDating,
	Updated ,
	Error
);
END_TYPE

// ---- DUTs/Motion/Axis Typ/Basic Typ/enumTyp/E_EncoderType.TcDUT
{attribute 'qualified_only'}
{attribute 'strict'}
TYPE E_EncoderType :
(
	Incremental := 0 ,
	Absolute := 1
);
END_TYPE

// ---- DUTs/Motion/Axis Typ/Basic Typ/Input/Basic_Input_typ.TcDUT
TYPE Basic_Input_typ : 	
	STRUCT 
		Command : Basic_Command_axis_typ;
		Parameter : Bacis_Parameter_axis_typ;
	END_STRUCT
END_TYPE

// ---- DUTs/Motion/Axis Typ/Basic Typ/Input/Cmd/Basic_Command_axis_typ.TcDUT
TYPE Basic_Command_axis_typ : 	
	STRUCT  (*command structure*)
		Power : BOOL; (*switch on the controller*)
		Home : BOOL; (*reference the axis*)
		MoveAbsolute : BOOL; (*move to an defined position*)
		MoveAdditive : BOOL; (*move a defiened distance*)
		MoveVelocity : BOOL; (*start a movement with a defiened velocity*)
		MoveRelative : BOOL;
		Halt : BOOL; (*stop every active movement*)
		Stop : BOOL; (*stop every active movement as long as is set*)
		MoveJogPos : BOOL; (*move in positive direction as long as is set*)
		MoveJogNeg : BOOL; (*move in negative direction as long as is set*)
		SetOverride : BOOL;
		pDriveAction:  POINTER TO PVOID; //enumDriveAction;
		ErrorAcknowledge : BOOL; (*reset active errors*)
		ClearFault: BOOL;
		AxisInit: 	BOOL;		
		MonitorDCEnable:	  BOOL;		
		MonitorTemperatureEnable: BOOL;
		LogEnable:	BOOL:=	TRUE;
				
	END_STRUCT
END_TYPE

// ---- DUTs/Motion/Axis Typ/Basic Typ/Input/Params/Bacis_Parameter_axis_typ.TcDUT
TYPE Bacis_Parameter_axis_typ : 	
	STRUCT  (*parameter structure*)
		ThreadName			: STRING[20];
		PosForLog			: REAL;//USINT;
		Position 			: LREAL; (*target-position for MoveAbsolute-Command*)
		Distance 			: LREAL; (*distance for MoveAdditive-Command*)
		Velocity 			: LREAL; (*velocity for MoveVelocity-Command*)
		Direction 			: MC_Direction ; (*direction for commanded movements*)
		Acceleration 		: LREAL; (*acceleration for commanded movements*)
		Deceleration 		: LREAL; (*deceleration for commanded movements*)
		EncoderOffset 		: DINT;
		JogVelocity 		: LREAL; (*velocity for jogging movement*)
		JogMod				: E_JogMode:= MC_JOGMODE_CONTINOUS;
		JogPosition			: LREAL ;//Relative distance for movements inMC_JOGMODE_INCHING mode
		HomeOptions         : ST_HomeOptions;
		Jerk 				: LREAL;
		Options 			: ST_MoveOptions ;
		BufferMode			: MC_BufferMode ;
		VelFactor 			: LREAL := 1.0; (*1.0 = 100% *)(*for Mc_SetOverride*)
		AccFactor 			: LREAL := 1.0; (*1.0 = 100% *)(*for Mc_SetOverride*)
		JerkFactor			: LREAL := 1.0; (*1.0 = 100% *)(*for Mc_SetOverride*)		
		pcNetId				: T_AmsNetID ; (* PC NetID*)		
		ecNetId				: T_AmsNetID ; (* EtherCAT NetID*)		
		ecNetIdArr			: T_AmsNetIdArr ; (* EtherCAT NetID*)		
		Drive				: Drive_Parameter_typ;		
		RatedCurrent 		: LREAL;
		Ratedtorque 		: LREAL;  //[Nm]
	//	MotorID             : eMotorID;
		pFlowID				: POINTER TO DINT;
	//	SubsysID			: eSubsystemID;
		Limits				: Motion_Limit_Parameter;
	END_STRUCT
END_TYPE

// ---- DUTs/Motion/Axis Typ/Basic Typ/Input/Params/Drive_Parameter_typ.TcDUT
TYPE Drive_Parameter_typ :
STRUCT
	eDriveType: 			enumDriveType;
	VendorNameID: 			eVendorNameID;
	EtherCatAddr: 			UINT ;
	sFoeParams_Path:		T_MaxString;
	sFoeFWFile_Path:		T_MaxString;	
	LatestParamVer:			UDINT;
	bDisableFoE_Transfer:	BOOL := TRUE;
	Kt:						LREAL	:= 1.0;	
END_STRUCT
END_TYPE

// ---- DUTs/Motion/Axis Typ/Basic Typ/Input/Params/Motion_Limit_Parameter.TcDUT
TYPE Motion_Limit_Parameter :
STRUCT	
	MaxTemperature: 	LREAL; 
	MinDC         : 	UDINT;
	MaxDC         : 	UDINT;
END_STRUCT
END_TYPE

// ---- DUTs/Motion/Axis Typ/Basic Typ/Input/Params/ST_BasicHomeParam.TcDUT
TYPE ST_BasicHomeParam :
STRUCT
	HomeMode: 			MC_HomingMode (*USINT*); 
	HomingOnDrive:      BOOL := FALSE;
	ExternalEncoder:    BOOL := FALSE;
	eEncoderType:		E_EncoderType;
	StartDirection: 	eHomeModeOption;	
	SwitchVelo: 		LREAL; 	//velovity that searching for the signal - Fast Velo
	TriggerVelo: 		LREAL ;	//velocity that move the axis to the configured switching edge - Slow Velo*)
	
	HomeSetPos: 		LREAL;
	AlignPos: 			LREAL;
	
	Jerk:				LREAL;	
	Acc:				LREAL;		 	 	
	Dcc:				LREAL;
END_STRUCT
END_TYPE

// ---- DUTs/Motion/Axis Typ/Basic Typ/Input/Params/ST_HomeAbsEncoder.TcDUT
TYPE ST_HomeAbsEncoder :
STRUCT
	
	BlockOffsetPosition: 	LREAL; 
END_STRUCT
END_TYPE

// ---- DUTs/Motion/Axis Typ/Basic Typ/Input/Params/ST_HomeAbsSwitch.TcDUT
TYPE ST_HomeAbsSwitch :
STRUCT
	pSignalInput		: POINTER TO BOOL;	
	SensorEdgeSignal 	: eHomeModeOption;	
	Trigger_Direction	: eHomeModeOption;
END_STRUCT
END_TYPE

// ---- DUTs/Motion/Axis Typ/Basic Typ/Input/Params/ST_HomeLagErr.TcDUT
TYPE ST_HomeLagErr :
STRUCT
	LagErr					: LREAL ;
	TriggerOffsetPos		: LREAL ;
	BlockSearchMaxCurrent	: INT;
	BlockExitMaxCurrent		: INT;
	BlockSearchRatedCurrent	: UDINT;
	BlockExitRatedCurrent	: UDINT;
	TorqueLimitPersent		: UINT;	//[%]
	BlockSearchPositionWindow : UDINT;	//[%]
	BlockExitPositionWindow	  : UDINT;
	
END_STRUCT
END_TYPE

// ---- DUTs/Motion/Axis Typ/Basic Typ/Input/Params/ST_HomeOptions.TcDUT
TYPE ST_HomeOptions :
STRUCT
	
	stBasic:		ST_BasicHomeParam;
	stLagErr:		ST_HomeLagErr;	
	stAbsSwitch:	ST_HomeAbsSwitch;
	 
END_STRUCT
END_TYPE

// ---- DUTs/Motion/Axis Typ/Basic Typ/Output/Basic_Error_axis_typ.TcDUT
TYPE Basic_Error_axis_typ : 	
	STRUCT 
		ErrorCount	: UINT ;
		fbErrorHandler : FB_ErrorHandler;	
	//	ErrorInfo : ERR_TASK_INFO_typ;
		ErrorEntry: Eh_ErrorEntry_typ;
	END_STRUCT
END_TYPE

// ---- DUTs/Motion/Axis Typ/Basic Typ/Output/Basic_Output_typ.TcDUT
TYPE Basic_Output_typ : 	
	STRUCT 
		monitor : Basic_Monitor_axis_typ;
		Status : Basic_Status_axis_typ;
		Error : Basic_Error_axis_typ;
	END_STRUCT
END_TYPE

// ---- DUTs/Motion/Axis Typ/Basic Typ/Output/Monitor/Basic_Monitor_axis_typ.TcDUT
TYPE Basic_Monitor_axis_typ : 	
	STRUCT 
		ActPosition : 		LREAL; (*actual position of the axis*)		
		ActVelocity :		LREAL; (*actual velocity of the axis*)
		SetVelocity:		LREAL;
		ActLagError : 		LREAL;
		ActualTorque : 		LREAL;
		ActualCurrent : 	LREAL;
		ModuloActPos : 		LREAL;
		SetPos:				LREAL;
		ModuloSetPos:		LREAL;
		SetVel:				LREAL;
		ActExternEncodPos 	AT %I* : UDINT;
		FileUpdate:			Basic_Monitor_FileUpdate_axis_typ;
		ActualDC  			: LREAL;// MilliAp
		stAbsEncoder:       ST_HomeAbsEncoder;
	END_STRUCT
END_TYPE

// ---- DUTs/Motion/Axis Typ/Basic Typ/Output/Monitor/Basic_Monitor_FileUpdate_axis_typ.TcDUT
TYPE Basic_Monitor_FileUpdate_axis_typ : 	
	STRUCT 

		FileUpdate_Error:	enum_DriveUpdateError;
		ErrorID: 			UDINT;
	END_STRUCT
END_TYPE

// ---- DUTs/Motion/Axis Typ/Basic Typ/Output/Status/Basic_MC_MoveVelocity_Status_typ.TcDUT
TYPE Basic_MC_MoveVelocity_Status_typ : 	
	STRUCT 
		In_Velocity : BOOL;
		Busy : BOOL;
		CommandAborted : BOOL;
		Active : BOOL ;
	END_STRUCT
END_TYPE

// ---- DUTs/Motion/Axis Typ/Basic Typ/Output/Status/Basic_MC_Power_Status_typ.TcDUT
TYPE Basic_MC_Power_Status_typ : 	
	STRUCT 
		Status : BOOL;
		Busy : BOOL;
	END_STRUCT
END_TYPE

// ---- DUTs/Motion/Axis Typ/Basic Typ/Output/Status/Basic_MC_Reset_Status_typ.TcDUT
TYPE Basic_MC_Reset_Status_typ : 
	STRUCT 
		Done : BOOL;
		Busy : BOOL;
	END_STRUCT
END_TYPE

// ---- DUTs/Motion/Axis Typ/Basic Typ/Output/Status/Basic_MC_SetOverride_typ.TcDUT
TYPE Basic_MC_SetOverride_typ : 	
	STRUCT 
		Enabled : BOOL;
		Busy : BOOL;
	END_STRUCT
END_TYPE

// ---- DUTs/Motion/Axis Typ/Basic Typ/Output/Status/Basic_Status_axis_typ.TcDUT
TYPE Basic_Status_axis_typ EXTENDS ReadStatus_typ : 	
	STRUCT 		
		FAULT 				: BOOL;
		DriveEnable 		: BOOL;     
		ReadyForCmd 		: BOOL;
		ClearFaultDone 		: BOOL;
		CommunicationError	: BOOL;
		MC_Power 			: Basic_MC_Power_Status_typ;
		MC_Home 			: Basic_Status_typ;
		MC_Reset 			: Basic_MC_Reset_Status_typ;
		MC_Halt 			: Basic_Status_typ;
		MC_Stop 			: Basic_Status_typ;
		MC_MoveAbsolut 		: Basic_Status_typ;
		MC_MoveAdditive 	: Basic_Status_typ;
		MC_MoveRelative		: Basic_Status_typ;
		MC_MoveVelocity 	: Basic_MC_MoveVelocity_Status_typ;
		MC_SetOverride 		: Basic_MC_SetOverride_typ;
		MC_Jog				: Basic_Status_typ ;
		AxisInitDone 		: BOOL;
		Drive				: Drive_Status_typ;
	END_STRUCT
END_TYPE

// ---- DUTs/Motion/Axis Typ/Basic Typ/Output/Status/Basic_Status_typ.TcDUT
TYPE Basic_Status_typ : 	
	STRUCT 
		Done : BOOL;
		Busy : BOOL;
		CommandAborted : BOOL;
		Active : BOOL ;
	END_STRUCT
END_TYPE

// ---- DUTs/Motion/Axis Typ/Basic Typ/Output/Status/Drive_Status_typ.TcDUT
TYPE Drive_Status_typ :
STRUCT
	ActiveHW:				BOOL;	
	eUpdate_Staus:			enum_DriveUpdateStatus;	
	ParamVer:				UDINT;
END_STRUCT
END_TYPE

// ---- DUTs/Motion/Axis Typ/Basic Typ/Output/Status/ReadStatus_typ.TcDUT
TYPE ReadStatus_typ :
STRUCT 
	AxisStatus             :ST_AxisStatus ;

END_STRUCT
END_TYPE

// ---- DUTs/Motion/Axis Typ/CyclicAxis_Typ/CyclicAxis_CMD_typ.TcDUT
TYPE CyclicAxis_CMD_typ :
STRUCT
		
	CyclicPos : CyclicPos_CMD_typ;
	CyclicVel : CyclicVel_CMD_typ;		
	
END_STRUCT
END_TYPE

// ---- DUTs/Motion/Axis Typ/CyclicAxis_Typ/CyclicAxis_Error_typ.TcDUT
TYPE CyclicAxis_Error_typ :
	STRUCT
		ErrorID : UDINT ;
		ErrorText : STRING[2048];(*ARRAY[0..3]OF STRING[79]*) (*Error Text*)
		ErrorEntry: Eh_ErrorEntry_typ;
	END_STRUCT
END_TYPE

// ---- DUTs/Motion/Axis Typ/CyclicAxis_Typ/CyclicAxis_Input_typ.TcDUT
TYPE CyclicAxis_Input_typ :
	STRUCT
		Command 	: CyclicAxis_CMD_typ ;
		Parameter	: CyclicAxis_Param_typ ;
	END_STRUCT
END_TYPE

// ---- DUTs/Motion/Axis Typ/CyclicAxis_Typ/CyclicAxis_monitor_typ.TcDUT
TYPE CyclicAxis_monitor_typ :
STRUCT
END_STRUCT
END_TYPE

// ---- DUTs/Motion/Axis Typ/CyclicAxis_Typ/CyclicAxis_Output_typ.TcDUT
TYPE CyclicAxis_Output_typ :
	STRUCT
		monitor 	: CyclicAxis_monitor_typ ;
		Status		: CyclicAxis_Status_typ ;
		Error		: CyclicAxis_Error_typ ;
		
	END_STRUCT
END_TYPE

// ---- DUTs/Motion/Axis Typ/CyclicAxis_Typ/CyclicAxis_Param_typ.TcDUT
TYPE CyclicAxis_Param_typ :
STRUCT
	
	ThreadName		: STRING[20];
	CyclicPos		: CyclicPos_Param_typ;
    CyclicVel		: CyclicVel_Param_typ;   
END_STRUCT
END_TYPE

// ---- DUTs/Motion/Axis Typ/CyclicAxis_Typ/CyclicAxis_Status_typ.TcDUT
TYPE CyclicAxis_Status_typ :
	STRUCT	
		CyclicPos:	CyclicPos_Status_typ;	
		CyclicVel:	CyclicVel_Status_typ;	
	END_STRUCT
END_TYPE

// ---- DUTs/Motion/Axis Typ/CyclicAxis_Typ/CyclicAxis_typ.TcDUT

TYPE CyclicAxis_typ :
	STRUCT
		Input	: CyclicAxis_Input_typ ;
		Output	: CyclicAxis_Output_typ ;
	END_STRUCT
END_TYPE

// ---- DUTs/Motion/Axis Typ/CyclicAxis_Typ/CyclicPos_CMD_typ.TcDUT
TYPE CyclicPos_CMD_typ :
STRUCT
	
	Start 		: BOOL;
	Disable 	: BOOL;
	
END_STRUCT
END_TYPE

// ---- DUTs/Motion/Axis Typ/CyclicAxis_Typ/CyclicPos_Param_typ.TcDUT
TYPE CyclicPos_Param_typ :
STRUCT
	
    SetPos			: LREAL;
	Velocity		: LREAL;
	MaxAcc			: LREAL;
	MaxDcc			: LREAL;
		
END_STRUCT
END_TYPE

// ---- DUTs/Motion/Axis Typ/CyclicAxis_Typ/CyclicPos_Status_typ.TcDUT
TYPE CyclicPos_Status_typ :
	STRUCT
		Active:		BOOL;	
		Busy:		BOOL;
	
	END_STRUCT
END_TYPE

// ---- DUTs/Motion/Axis Typ/CyclicAxis_Typ/CyclicVel_CMD_typ.TcDUT
TYPE CyclicVel_CMD_typ :
STRUCT
	
	Start 		: BOOL;
	Disable 	: BOOL;
	
END_STRUCT
END_TYPE

// ---- DUTs/Motion/Axis Typ/CyclicAxis_Typ/CyclicVel_Param_typ.TcDUT
TYPE CyclicVel_Param_typ :
STRUCT
    SetVel			: LREAL;
	MaxVelocity		: LREAL;
	MaxAcc			: LREAL;
	MaxDcc			: LREAL;
	Jerk			: LREAL;
END_STRUCT
END_TYPE

// ---- DUTs/Motion/Axis Typ/CyclicAxis_Typ/CyclicVel_Status_typ.TcDUT
TYPE CyclicVel_Status_typ :
	STRUCT
		Active:		BOOL;	
		Busy:		BOOL;
	
	END_STRUCT
END_TYPE

// ---- DUTs/Motion/Axis Typ/CyclicAxis_Typ/eCyclicAxisState.TcDUT
TYPE eCyclicAxisState :
	(
		CyclicAxis_STATE_WAIT := 0,
		CyclicAxis_STATE_READY,
		CyclicAxis_STATE_START,
		CyclicAxis_STATE_DISABLE,		
		CyclicAxis_STATE_POS_ACTIVE,
		CyclicAxis_STATE_VEL_ACTIVE,
		CyclicAxis_STATE_ERROR
	);
END_TYPE

// ---- DUTs/Motion/Axis Typ/ExtendedAxisTyp_1.TcDUT
TYPE ExtendedAxisTyp_1  :
	STRUCT
		Basic_axis 	: Basic_axis_typ;
		MultiAxis 	: MultiAxis_typ;
		CyclicAxis	: CyclicAxis_typ;
		ParIDAccess	: ParIDAccess_Typ;
		VelocityCtrl: VelocityCtrl_typ;
	END_STRUCT
END_TYPE

// ---- DUTs/Motion/Axis Typ/MultiAxis_Typ/CamIn_CMD_typ.TcDUT
TYPE CamIn_CMD_typ :
STRUCT
	StartSlave : BOOL ;
	DisengageSlave : BOOL ;
END_STRUCT
END_TYPE

// ---- DUTs/Motion/Axis Typ/MultiAxis_Typ/CamIn_Param_typ.TcDUT
TYPE CamIn_Param_typ :
	STRUCT
		MasterOffset 	:	LREAL:=			1.0;
		SlaveOffset 	:	LREAL:=			1.0;
		MasterScaling 	:	LREAL:= 		1.0;
		SlaveScaling 	: 	LREAL:= 		1.0;
		StartMode 		: 	MC_StartMode:=	MC_STARTMODE_RELATIVE;
		CamTableID 		: 	MC_CAM_ID:=		123; 
		BufferMode 		:	MC_BufferMode; 
		Options 		: 	ST_CamInOptions;

	END_STRUCT
END_TYPE

// ---- DUTs/Motion/Axis Typ/MultiAxis_Typ/CamIn_Statuses_typ.TcDUT
TYPE CamIn_Statuses_typ :
	STRUCT
		InSync 			: 		BOOL;
		Busy 			: 		BOOL; 
		Active 			: 		BOOL; 
		CommandAborted 	: 		BOOL;

	END_STRUCT
END_TYPE

// ---- DUTs/Motion/Axis Typ/MultiAxis_Typ/CamOut_Param_typ.TcDUT
TYPE CamOut_Param_typ :
	STRUCT
		Options 		: ST_GearOutOptions; //Currently not implemented/used
	END_STRUCT
END_TYPE

// ---- DUTs/Motion/Axis Typ/MultiAxis_Typ/CamOut_Statuses_typ.TcDUT
TYPE CamOut_Statuses_typ EXTENDS MultiAxis_Status_typ :
STRUCT
END_STRUCT
END_TYPE

// ---- DUTs/Motion/Axis Typ/MultiAxis_Typ/CamTableSelectCMD_typ.TcDUT
TYPE CamTableSelectCMD_typ :
	STRUCT
		
		Start 		: BOOL;

	END_STRUCT
END_TYPE

// ---- DUTs/Motion/Axis Typ/MultiAxis_Typ/CamTableSelect_Param_typ.TcDUT
TYPE CamTableSelect_Param_typ :
	STRUCT
	    Periodic 		: BOOL; 
		MasterAbsolute 	: BOOL; 
		SlaveAbsolute 	: BOOL; 
		CamTableID 		: MC_CAM_ID;
		CamTable 		: MC_CAM_REF; // can have  ARRAY[1..n] OF MC_MotionFunctionPoint or Table1 : ARRAY[0..360, 0..1] OF LREAL

	END_STRUCT
END_TYPE

// ---- DUTs/Motion/Axis Typ/MultiAxis_Typ/CamTableSelect_Status_typ.TcDUT
TYPE CamTableSelect_Status_typ EXTENDS MultiAxis_Status_typ :
	STRUCT
		
	END_STRUCT
END_TYPE

// ---- DUTs/Motion/Axis Typ/MultiAxis_Typ/eMultiAxisState.TcDUT
TYPE eMultiAxisState :
	(
		MultiAxis_STATE_WAIT := 0,
		MultiAxis_STATE_ENTER_READY,
		MultiAxis_STATE_READY,		
		MultiAxis_STATE_GEAR_START,
		MultiAxis_STATE_GEAR_STOP,
		MultiAxis_STATE_CAM_SELECT,
		MultiAxis_STATE_CAM_START,
		MultiAxis_STATE_CAM_STOP,
		MultiAxis_STATE_GEAR_IN_DYN,
		MultiAxis_STATE_GEAR_IN_POS,
		MultiAxis_STATE_GEAR_OUT,
		MultiAxis_STATE_GEAR_IN_MULTI_MASTER,
	
		MultiAxis_STATE_ERROR
	);
END_TYPE

// ---- DUTs/Motion/Axis Typ/MultiAxis_Typ/GearInDyn_CMD_typ.TcDUT
TYPE GearInDyn_CMD_typ :
STRUCT
	StartSlave : BOOL ;
	DisengageSlave : BOOL ;
END_STRUCT
END_TYPE

// ---- DUTs/Motion/Axis Typ/MultiAxis_Typ/GearInDyn_Param_typ.TcDUT
TYPE GearInDyn_Param_typ :
	STRUCT
		GearRatio    : LREAL;   
		Acceleration : LREAL;   
		Deceleration : LREAL;   
		Jerk         :LREAL;   
		BufferMode   :MC_BufferMode;   //Currently not implemented
		Options      :ST_GearInDynOptions;//Currently not implemented

	END_STRUCT
END_TYPE

// ---- DUTs/Motion/Axis Typ/MultiAxis_Typ/GearInDyn_Statuses_typ.TcDUT
TYPE GearInDyn_Statuses_typ :
	STRUCT
		InGear 			: 		BOOL;
		Busy 			: 		BOOL; 
		Active 			: 		BOOL; 
		CommandAborted 	: 		BOOL;

	END_STRUCT
END_TYPE

// ---- DUTs/Motion/Axis Typ/MultiAxis_Typ/GearInMultiMaster_CMD_typ.TcDUT
TYPE GearInMultiMaster_CMD_typ :
STRUCT
	StartSlave : BOOL ;
	DisengageSlave : BOOL ;
END_STRUCT
END_TYPE

// ---- DUTs/Motion/Axis Typ/MultiAxis_Typ/GearInMultiMaster_Param_typ.TcDUT
TYPE GearInMultiMaster_Param_typ :
	STRUCT
	GearRatio1  	: LREAL;
    GearRatio2   	: LREAL;
    GearRatio3   	: LREAL;
    GearRatio4   	: LREAL;
    Acceleration 	: LREAL;
    Deceleration 	: LREAL;
    Jerk         	: LREAL;
    BufferMode   	: MC_BufferMode;
    Options      	: ST_GearInMultiMasterOptions;

	END_STRUCT
END_TYPE

// ---- DUTs/Motion/Axis Typ/MultiAxis_Typ/GearInMultiMaster_Statuses_typ.TcDUT
TYPE GearInMultiMaster_Statuses_typ :
	STRUCT
		InGear 			: 		BOOL;
		Busy 			: 		BOOL; 
		Active 			: 		BOOL; 
		CommandAborted 	: 		BOOL;
	END_STRUCT
END_TYPE

// ---- DUTs/Motion/Axis Typ/MultiAxis_Typ/GearInPos_CMD_typ.TcDUT
TYPE GearInPos_CMD_typ :
STRUCT
	StartSlave : BOOL ;
	DisengageSlave : BOOL ;
END_STRUCT
END_TYPE

// ---- DUTs/Motion/Axis Typ/MultiAxis_Typ/GearInPos_Param_typ.TcDUT
TYPE GearInPos_Param_typ :
	STRUCT
		RatioNumerator   	: LREAL  := 1;
        RatioDenominator   	: UINT   := 1;
        MasterSyncPosition 	: LREAL;     (* absolute master synchronous position *)
        SlaveSyncPosition  	: LREAL;     (* absolute slave synchronous position *)
        SyncMode           	: ST_SyncMode;//The boundary conditions for the synchronisation are specified in the SyncMode variables
		MasterStartDistance	: LREAL;
        Velocity           	: LREAL := 0; //Maximum slave velocity in the synchronisation phase. If a velocity is not specified, the maximum velocity of the axis from the system manager data is used.
        Acceleration       	: LREAL; //Maximum slave acceleration in the synchronisation phase   (* 0 : use default value *)
        Deceleration       	: LREAL; //Maximum slave deceleration in the synchronisation phase    (* 0 : use default value *)
        Jerk               	: LREAL; //Maximum slave jerk in the synchronisation phase    (* 0 : use default value *)
		BufferMode   		:MC_BufferMode;   //Currently not implemented
		Options      		:ST_GearInDynOptions;//Currently not implemented	
	END_STRUCT
END_TYPE

// ---- DUTs/Motion/Axis Typ/MultiAxis_Typ/GearInPos_Statuses_typ.TcDUT
TYPE GearInPos_Statuses_typ :
	STRUCT
		StartSync       : BOOL;
        InSync          : BOOL;
        CommandAborted  : BOOL;
		Active 			: BOOL;
		Busy			: BOOL;

	END_STRUCT
END_TYPE

// ---- DUTs/Motion/Axis Typ/MultiAxis_Typ/GearOut_Param_typ.TcDUT
TYPE GearOut_Param_typ :
	STRUCT
		Options : ST_GearOutOptions; // Currently not implemented

	END_STRUCT
END_TYPE

// ---- DUTs/Motion/Axis Typ/MultiAxis_Typ/GearOut_Statuses_typ.TcDUT
TYPE GearOut_Statuses_typ EXTENDS MultiAxis_Status_typ:
	STRUCT
		

	END_STRUCT
END_TYPE

// ---- DUTs/Motion/Axis Typ/MultiAxis_Typ/MultiAxis_CMD_typ.TcDUT
TYPE MultiAxis_CMD_typ :
	STRUCT		
		CamTableSelect		: CamTableSelectCMD_typ ;
		CamIn				: CamIn_CMD_typ ;
		GearInDyn			: GearInDyn_CMD_typ ;
		GearInPos			: GearInPos_CMD_typ ;
		GearInMultiMaster 	: GearInMultiMaster_CMD_typ ;
	END_STRUCT
END_TYPE

// ---- DUTs/Motion/Axis Typ/MultiAxis_Typ/MultiAxis_Error_typ.TcDUT
TYPE MultiAxis_Error_typ :
	STRUCT
		ErrorID : UDINT ;
		ErrorText : STRING[2048];(*ARRAY[0..3]OF STRING[79]*) (*Error Text*)
	END_STRUCT
END_TYPE

// ---- DUTs/Motion/Axis Typ/MultiAxis_Typ/MultiAxis_Input_typ.TcDUT
TYPE MultiAxis_Input_typ :
	STRUCT
		Command 	: MultiAxis_CMD_typ ;
		Parameter	: MultiAxis_Param_typ ;
	END_STRUCT
END_TYPE

// ---- DUTs/Motion/Axis Typ/MultiAxis_Typ/MultiAxis_monitor_typ.TcDUT
TYPE MultiAxis_monitor_typ :
STRUCT
END_STRUCT
END_TYPE

// ---- DUTs/Motion/Axis Typ/MultiAxis_Typ/MultiAxis_Output_typ.TcDUT
TYPE MultiAxis_Output_typ :
	STRUCT
		monitor 	: MultiAxis_monitor_typ ;
		Status		: MultiAxis_Statuses_typ ;
		Error		: MultiAxis_Error_typ ;
		
	END_STRUCT
END_TYPE

// ---- DUTs/Motion/Axis Typ/MultiAxis_Typ/MultiAxis_Param_typ.TcDUT
TYPE MultiAxis_Param_typ :
	STRUCT
		ThreadName			: STRING[20];
		CamTableSelect		: CamTableSelect_Param_typ ;
		CamIn				: CamIn_Param_typ ;
		CamOut				: CamOut_Param_typ ;
		GearInDyn			: GearInDyn_Param_typ ;
		GearInPos			: GearInPos_Param_typ ;
		GearOut				: GearOut_Param_typ ;
		GearInMultiMaster	: GearInMultiMaster_Param_typ ;
	END_STRUCT
END_TYPE

// ---- DUTs/Motion/Axis Typ/MultiAxis_Typ/MultiAxis_Statuses_typ.TcDUT
TYPE MultiAxis_Statuses_typ :
	STRUCT
		CamTableSelect  	: CamTableSelect_Status_typ ;
		CamIn 				: CamIn_Statuses_typ ;
		CamOut				: CamOut_Statuses_typ ;
		GearInDyn			: GearInDyn_Statuses_typ ;
		GearInPos			: GearInPos_Statuses_typ ;
		GearOut				: GearOut_Statuses_typ ;	
		GearInMultiMaster 	: GearInMultiMaster_Statuses_typ;	
	END_STRUCT
END_TYPE

// ---- DUTs/Motion/Axis Typ/MultiAxis_Typ/MultiAxis_Status_typ.TcDUT
TYPE MultiAxis_Status_typ :
	STRUCT
		Done  		: BOOL;
		Busy 		: BOOL;
	END_STRUCT
END_TYPE

// ---- DUTs/Motion/Axis Typ/MultiAxis_Typ/MultiAxis_typ.TcDUT
TYPE MultiAxis_typ :
	STRUCT
		Input	: MultiAxis_Input_typ ;
		Output	: MultiAxis_Output_typ ;
	END_STRUCT
END_TYPE

// ---- DUTs/Motion/Axis Typ/ParIDAccess_Typ/eParIDAccessState.TcDUT
TYPE eParIDAccessState :
	(
		ParID_STATE_WAIT := 0,
		ParID_STATE_READY,
		ParID_STATE_READ_SDO,
		ParID_STATE_WRITE_SDO,		
		ParID_STATE_ERROR
	);
END_TYPE

// ---- DUTs/Motion/Axis Typ/ParIDAccess_Typ/ParIDAccess_CMD_typ.TcDUT
TYPE ParIDAccess_CMD_typ :
STRUCT
		
	WriteCoeSdo : BOOL;
	ReadCoeSdo : BOOL;	
	
END_STRUCT
END_TYPE

// ---- DUTs/Motion/Axis Typ/ParIDAccess_Typ/ParIDAccess_Error_typ.TcDUT
TYPE ParIDAccess_Error_typ :
	STRUCT
		ErrorID : UDINT ;
		ErrorText : STRING[2048];(*ARRAY[0..3]OF STRING[79]*) (*Error Text*)
		ErrorEntry: Eh_ErrorEntry_typ;
	END_STRUCT
END_TYPE

// ---- DUTs/Motion/Axis Typ/ParIDAccess_Typ/ParIDAccess_Input_typ.TcDUT
TYPE ParIDAccess_Input_typ :
	STRUCT
		Command 	: ParIDAccess_CMD_typ ;
		Parameter	: ParIDAccess_Param_typ ;
	END_STRUCT
END_TYPE

// ---- DUTs/Motion/Axis Typ/ParIDAccess_Typ/ParIDAccess_monitor_typ.TcDUT
TYPE ParIDAccess_monitor_typ :
STRUCT
END_STRUCT
END_TYPE

// ---- DUTs/Motion/Axis Typ/ParIDAccess_Typ/ParIDAccess_Output_typ.TcDUT
TYPE ParIDAccess_Output_typ :
	STRUCT
		monitor 	: ParIDAccess_monitor_typ ;
		Status		: ParIDAccess_Status_axis_typ ;
		Error		: ParIDAccess_Error_typ ;
		
	END_STRUCT
END_TYPE

// ---- DUTs/Motion/Axis Typ/ParIDAccess_Typ/ParIDAccess_Param_typ.TcDUT
TYPE ParIDAccess_Param_typ :
STRUCT
	
	ThreadName		: STRING[20];
	WriteCoeSdo	: ParIDAccess_Par_WriteCoedSdo_typ;
	ReadCoedSdo	: ParIDAccess_Par_ReadCoedSdo_typ;
	
END_STRUCT
END_TYPE

// ---- DUTs/Motion/Axis Typ/ParIDAccess_Typ/ParIDAccess_Par_ReadCoedSdo_typ.TcDUT
TYPE ParIDAccess_Par_ReadCoedSdo_typ : 	
	STRUCT  (*parameter structure*)
		
        nSubIndex       : BYTE; 
        nIndex          : WORD;
		pDstBuf         : POINTER TO DWORD; 
		cbBufLen        : UDINT; 
		tTimeout        : TIME := DEFAULT_ADS_TIMEOUT; 

	END_STRUCT
END_TYPE

// ---- DUTs/Motion/Axis Typ/ParIDAccess_Typ/ParIDAccess_Par_WriteCoedSdo_typ.TcDUT
TYPE ParIDAccess_Par_WriteCoedSdo_typ : 	
	STRUCT  (*parameter structure*)
		
        nSubIndex       : BYTE; 
        nIndex          : WORD;
        pSrcBuf         : POINTER TO DWORD; 
        cbBufLen        : UDINT; 
        tTimeout        : TIME := DEFAULT_ADS_TIMEOUT ;

	END_STRUCT
END_TYPE

// ---- DUTs/Motion/Axis Typ/ParIDAccess_Typ/ParIDAccess_Status_axis_typ.TcDUT
TYPE ParIDAccess_Status_axis_typ :
	STRUCT	
		WriteCoeSdo			: ParIDAccess_Status_typ ;
		ReadCoeSdo			: ParIDAccess_Status_typ ;	
	END_STRUCT
END_TYPE

// ---- DUTs/Motion/Axis Typ/ParIDAccess_Typ/ParIDAccess_Status_typ.TcDUT
TYPE ParIDAccess_Status_typ : 	
	STRUCT 
		Done : BOOL;
		Busy : BOOL;
		CommandAborted : BOOL;
		Active : BOOL ;
	END_STRUCT
END_TYPE

// ---- DUTs/Motion/Axis Typ/ParIDAccess_Typ/ParIDAccess_Typ.TcDUT
TYPE ParIDAccess_Typ :
STRUCT
	Input	: ParIDAccess_Input_typ ;
	Output	: ParIDAccess_Output_typ ;
END_STRUCT
END_TYPE

// ---- DUTs/Motion/Axis Typ/stAxisIF.TcDUT
TYPE stAxisIF :
STRUCT
END_STRUCT
END_TYPE

// ---- DUTs/Motion/Axis Typ/VelocityCtrl/eTorqueMode.TcDUT
TYPE eTorqueMode :
	(		
		mcFF :=0 ,
		mcLimit 
		
	);
END_TYPE

// ---- DUTs/Motion/Axis Typ/VelocityCtrl/eVelocityCtrlState.TcDUT
TYPE eVelocityCtrlState :
	(		
		VELOCITY_CTRL_STATE_WAIT :=0 ,
		VELOCITY_CTRL_STATE_READY :=1,					
		VELOCITY_CTRL_CNG_TO_VEL_MODE :=2,
		VELOCITY_CTRL_READ_POS_CTRL_VALUES :=3,
		VELOCITY_CTRL_MOVE_VELOCITY :=4,
		VELOCITY_CTRL_WAIT_MOVE_VELOCITY_DONE := 5,
		VELOCITY_CTRL_ACTIVE :=6,
		VELOCITY_CTRL_ACTIVE_STAND_STILL :=7,		
		VELOCITY_CTRL_InitSctrl :=8,
		VELOCITY_CTRL_CHANGE_TORQUE :=9,		
		VELOCITY_CTRL_STATE_STOP :=10 ,
		VELOCITY_CTRL_STATE_RETURN_ORG_VALUES := 11,
		VELOCITY_CTRL_DISABLE  :=12,		
		VELOCITY_CTRL_STATE_ERROR := 13,
		VELOCITY_CTRL_STEP_BY_STEP_STATE :=14,
		VELOCITY_CTRL_STEP_BY_STEP_STATE2 :=15
		
		
	);
END_TYPE

// ---- DUTs/Motion/Axis Typ/VelocityCtrl/VelocityCtrl_CMD_typ.TcDUT
TYPE VelocityCtrl_CMD_typ :
STRUCT
		

		Enable       : BOOL;		// Enable to exit set enable false		 
		InitSctrl    : BOOL;		// init pid
		Stop         : BOOL;		// Stop motor. stay in velocity control	
		
		//
	
		
END_STRUCT
END_TYPE

// ---- DUTs/Motion/Axis Typ/VelocityCtrl/VelocityCtrl_Error_typ.TcDUT
TYPE VelocityCtrl_Error_typ :
	STRUCT
		ErrorID : UDINT ;
		ErrorText : STRING[2048];(*ARRAY[0..3]OF STRING[79]*) (*Error Text*)
		ErrorEntry: Eh_ErrorEntry_typ;
	END_STRUCT
END_TYPE

// ---- DUTs/Motion/Axis Typ/VelocityCtrl/VelocityCtrl_Input_typ.TcDUT
TYPE VelocityCtrl_Input_typ :
	STRUCT
		Command 	: VelocityCtrl_CMD_typ ;
		Parameter	: VelocityCtrl_Param_typ ;
	END_STRUCT
END_TYPE

// ---- DUTs/Motion/Axis Typ/VelocityCtrl/Velocityctrl_monitor_typ.TcDUT
TYPE Velocityctrl_monitor_typ :
STRUCT
	OrgVelKp        			: LREAL;
	SetCyclicTorque 			: LREAL;
	OrgMaxTorque 				: LREAL;				
	OrgCyclicTorque 			: LREAL;			
	OrgSctrlKp 					: LREAL;
	OrgSctrlKi 					: LREAL;
	OrgGainCtrl 				: LREAL;
	OrgAccToCloseThePosError 	:LREAL; 
END_STRUCT
END_TYPE

// ---- DUTs/Motion/Axis Typ/VelocityCtrl/VelocityCtrl_Output_typ.TcDUT
TYPE VelocityCtrl_Output_typ :
	STRUCT
		monitor 	: Velocityctrl_monitor_typ ;
		Status		: VelocityCtrl_Status_typ ;
		Error		: VelocityCtrl_Error_typ ;
		
	END_STRUCT
END_TYPE

// ---- DUTs/Motion/Axis Typ/VelocityCtrl/VelocityCtrl_Param_typ.TcDUT
TYPE VelocityCtrl_Param_typ : 	
	STRUCT  (*parameter structure*)
		
		CyclicVelocity : LREAL;
		CyclicVelocityCorrection : REAL;
		CyclicTorque : LREAL;		
		Acceleration : LREAL := 1000000;
		Deceleration : LREAL := 2000000;
		SctrlKp 	 : LREAL  ; // 1/1000
		SctrlKi 	 : LREAL;	// 1/1000
		TorqueMode: eTorqueMode;
		ThreadName		: STRING[20]; 
		
	END_STRUCT
END_TYPE

// ---- DUTs/Motion/Axis Typ/VelocityCtrl/VelocityCtrl_Status_typ.TcDUT
TYPE VelocityCtrl_Status_typ : 	
	STRUCT 
		Done	   : BOOL;
		SctrlInitialized : BOOL;
		UpdateTorqueDone : BOOL;
		Busy       : BOOL;
		CommandAborted : BOOL;
		Active : BOOL ;
		InStopVelCtrl : BOOL ;
	END_STRUCT
END_TYPE

// ---- DUTs/Motion/Axis Typ/VelocityCtrl/VelocityCtrl_typ.TcDUT

TYPE VelocityCtrl_typ :
	STRUCT
		Input	: VelocityCtrl_Input_typ ;
		Output	: VelocityCtrl_Output_typ ;
	END_STRUCT
END_TYPE

// ---- DUTs/Motion/CoE_Obj_typ.TcDUT
TYPE CoE_Obj_typ :
STRUCT
	Index  	 : WORD;
	SunIndex : BYTE;
	Size	 : UDINT;   
	IsReal 	 : BOOL;  

END_STRUCT
END_TYPE

// ---- DUTs/Motion/Enums/eMotorID.TcDUT
{attribute 'qualified_only'}
//{attribute 'strict'}
{attribute 'to_string'}
TYPE eMotorID :
(
	NoMotor := 	0,
	ITM ,
	BKT_TensionFront ,
	BKT_TensionRear ,
	BKT_LateralFront ,
	BKT_LateralRear ,
	BKT_HeaterLowerAirKnivesBlower ,
	BKT_HeaterUpperAirKnivesBlower ,
	BlanketEngageFrontValve_1 ,
	BlanketEngageFrontValve_2 ,
	BlanketEngageFrontValve_3 ,
	BlanketEngageFrontValve_4 ,
	BlanketEngageFrontValve_5 ,
	BlanketEngageFrontValve_6 ,
	BlanketEngageRearValve_1 ,
	BlanketEngageRearValve_2 ,
	BlanketEngageRearValve_3 ,
	BlanketEngageRearValve_4 ,
	BlanketEngageRearValve_5 ,
	BlanketEngageRearValve_6 ,
	BKT_FeedSupportRoller ,
	BKT_EdgeSensorFan ,
	BKT_IndexSensorFan ,
	BKT_RegCamerasCoolingValve ,
	BRU_StickyRotate ,
	BRU_StickyEngageFront ,
	BRU_StickyEngageRear ,
	BRU_Heater ,
	BRU_StickyPeeling ,
	BRU_StickyServiceDisengage ,
	BRU_BWS ,
	BWS_MiteringPump ,
	BWS_CirculationPump ,	
	ASID_Drive ,
	ChargeRollerEngage ,
	LPH_EngageFront ,
	LPH_EngageRear ,
	LPH_CoolingValve ,
	LPH_CoolingPump ,
	LPH_CoolingTankHeater ,
	CS_WettingRoller ,
	CS_CollectingRoller ,
	CS_Engage ,
	CS_Disengage ,
	CR_Engage ,
	BID_Drive ,
	BID_EngageFront ,
	BID_EngageRear ,
	INK_ChargeDirectorPump ,
	INK_to_BID_pump ,
	INK_RDU_Valve ,
	INK_ExtractionPistonDown ,
	INK_ExtractionPistonUp ,
	INK_TubeEngageValve ,
	INK_TubeDisengageValve ,
	INK_TubeSliderPiston ,
	INK_RevolverLiftValve ,
	UW_Roller ,
	UW_ArmsUp ,
	UW_ArmsDown ,
	UW_RightClamp ,
	UW_LeftClamp ,
	UW_WebGuide ,
	WHS_FI ,
	WHS_PTR ,
	WHS_IPE_Front ,
	WHS_IPE_Rear ,
	WHS_IMP ,
	WHS_Peeler ,
	WHS_FP ,
	WHS_FE ,
	WHS_FI_NipEngageValve ,
	WHS_FI_NipDisengageValve ,
	WHS_FR_NipValve ,
	WHS_FP_NipEngageValve ,
	WHS_FP_NipDisengageValve ,
	WHS_FE_NipEngageValve ,
	WHS_FE_NipDisengageValve ,
	WHS_PE_WebGuide ,
	WHS_IBS ,
	WHS_BRI ,
	WHS_BRO ,
	WHS_ReinsertionXposition  ,
	RW_Roller ,
	RW_RightClamp,
	RW_LeftClamp ,
	RW_AirShaft ,
	RW_PackerArm  ,
	SPM_X ,
	SPM_Z ,
	ILP_FI_Motor ,
	ILP_FI_Nip ,
	ILP_FB_Motor ,
	ILP_FB_NipEngage ,
	PrimingMotor ,
	PrimingPump ,
	PrimerInputValve ,
	PrimerOutputValve ,
	DrainValve ,
	LowerRubberRollerEngage ,
	UpperRubberRollerEngage ,
	ImpressionEngage ,
	ILP_DryerBlower ,
	ILP_DryerExhaust ,
	ILP_DryerHeater ,
	ILP_FastCoolingValve ,
	ILP_CORONA_Ozone_Suction ,
	CVC1A_CoolingBlower ,
	CVC1B_CoolingBlower ,
	CVC2A_CoolingBlower ,
	CVC2B_CoolingBlower ,
	CVC_WaterPump ,
	CVC_WaterSupply  ,
	CVC_WaterReturn ,
	CVC_HX_WaterValve ,
	IMO_CS_CoolingHigh_1 ,
	IMO_CS_CoolingHigh_2 ,
	IMO_CS_CoolingHigh_3 ,
	IMO_CS_CoolingHigh_4 ,
	IMO_CS_CoolingHigh_5 ,
	IMO_CS_CoolingHigh_6 ,
	IMO_CS_CoolingMid_1 ,
	IMO_CS_CoolingMid_2 ,
	IMO_CS_CoolingMid_3 ,
	IMO_CS_CoolingMid_4 ,
	IMO_CS_CoolingMid_5 ,
	IMO_CS_CoolingMid_6 ,
	IMO_CS_CoolingLow_1 ,
	IMO_CS_CoolingLow_2 ,
	IMO_CS_CoolingLow_3 ,
	IMO_CS_CoolingLow_4 ,
	IMO_CS_CoolingLow_5 ,
	IMO_CS_CoolingLow_6 ,
	IMO_CS_InletPump_1 ,
	IMO_CS_InletPump_2 ,
	IMO_CS_InletPump_3 ,
	IMO_CS_InletPump_4 ,
	IMO_CS_InletPump_5 ,
	IMO_CS_InletPump_6 ,
	IMO_CS_ReturnPump ,
	IMO_EFS_Motor ,
	IMO_EFS_FilterPump ,
	IMO_PE_WastePump ,
	IMO_UC_WastePump ,
	IWS_WaterPumpRight,
	IWS_WaterPumpLeft,
	IWS_InputValveRight,	
	IWS_InputValveLeft,	
	IWS_InkWaterValve_1,	
	IWS_InkWaterValve_2,	
	IWS_InkWaterValve_3,	
	IWS_InkWaterValve_4,	
	IWS_InkWaterValve_5,	
	IWS_InkWaterValve_6,	
	IWS_InkWaterValve_7,	
	IWS_InkWaterValve_8,	
	IWS_InkWaterValve_9,	
	IWS_InkWaterValve_10,	
	IWS_InkWaterValve_11,	
	IWS_InkWaterValve_12,	
	UC_EC_Fans_1 ,
	UC_EC_Fans_2 ,
	UC_EC_Fans_3 ,
	UC_EC_Fans_4 ,
	LAST 
)DINT;
END_TYPE

// ---- DUTs/Motion/Enums/eSensorID.TcDUT
{attribute 'qualified_only'}
//{attribute 'strict'}
{attribute 'to_string'}
TYPE eSensorID :
(
	NoSensor,
	BKT_EDGE_SNS,
	BKT_IND_NPN_SNS,
	BKT_IND_PNP_SNS, 
	BKT_TENS_FRNT_HOME_SNS, 
	BKT_TENS_RR_HOME_SNS,
	BKT_TENS_FRNT_LD_CELL,
	BKT_TENS_RR_LD_CELL,
	BKT_TENS_SAFE_DETCT,
	BKT_LTRL_FRNT_HOME_SNS,
	BKT_LTRL_RR_HOME_SNS,
	SUP_ROLL_HOME_SNS,
	BRU_STKY_PEEL_HOME_SNS,
	BRU_STKY_MID_ROLLER_SNS,
	BRU_STKY_STIR_IN_PLC_SNS,
	BRU_STKY_TRAY_LVL_MID,
	BRU_STKY_TRAY_LVL_TOP,
	BRU_STKY_MID_ROL_TEMP,
	BRU_BWS_IN_PLC_SNS,
	BRU_BWS_FRNT_LIMT_SNS,
	BRU_BWS_RR_LIMT_SNS,
	BRU_BWS_LVL_SW_TOP,
	BRU_BWS_LVL_SW_BOT,
	BRT_SRV_POS_FRNT_1,
	BRT_SRV_POS_FRNT_2,
	BRT_SRV_POS_FRNT_3,
	BRT_SRV_POS_FRNT_4,
	BRT_SRV_POS_FRNT_5,
	BRT_SRV_POS_FRNT_6,
	BRT_SRV_POS_RR_1,
	BRT_SRV_POS_RR_2,
	BRT_SRV_POS_RR_3,
	BRT_SRV_POS_RR_4,
	BRT_SRV_POS_RR_5,
	BRT_SRV_POS_RR_6,
	EH_TMP_SNS_01,
	EH_TMP_SNS_02,
	EH_TMP_SNS_03,
	EH_TMP_SNS_04,
	EH_TMP_SNS_05,
	EH_TMP_SNS_06,
	EH_TMP_SNS_07A,
	EH_TMP_SNS_07B,
	EH_TMP_SNS_08,
	EH_TMP_SNS_09,
	EH_TMP_SNS_10A,
	EH_TMP_SNS_10B,
	EH_HOOD_IN_PLC_SNS_07,
	EH_HOOD_IN_PLC_SNS_08,
	EH_HOOD_IN_PLC_SNS_09,
	EH_HOOD_IN_PLC_SNS_10,
	EH_SUC_PRSSR_SNS_01,
	EH_SUC_PRSSR_SNS_02,
	EH_SUC_PRSSR_SNS_03,
	EH_SUC_PRSSR_SNS_04,
	EH_SUC_PRSSR_SNS_05,
	EH_SUC_PRSSR_SNS_06,
	EH_SUC_PRSSR_SNS_07,
	EH_SUC_PRSSR_SNS_08,
	EH_SUC_PRSSR_SNS_09,
	EH_SUC_PRSSR_SNS_10,
	EH_TOP_AIR_KNF_PRSSR_SNS,
	EH_BTM_AIR_KNF_PRSSR_SNS,
	EH_TOP_AIR_KNF_BLWR_TMP,
	EH_BTM_AIR_KNF_BLWR_TMP,
	EH_AIR_PRG_PRSSR_SNS,
	ITM_DRUM_FRNT_TEMP_SNS, 
	ITM_DRUM_RR_TEMP_SNS,
	EBV_SUC_PRS_SNS,
	EBV_TEMP_SNS,
	ITC_TMP_SNS,
	ITC_LVL_SNS,
	ASID_IN_PLC_SNS,
	ASID_DRUM_TEMP_SNS,
	ASID_DRV_TEMP,
	CR_IN_PLC_SNS,
	CR_DISENG_FRT_SNS,
	CR_DISENG_RR_SNS,
	ELECTROMETER_OUT,
	CS_IN_PLC_SNS,
	CS_ENG_SNS,
	CS_DISENG_SNS,
	CS_AIR_PRSR_SNS,
	CS_TEMP_SNS,
	BID_1A_FLD_IN_PLACE_SNS,
	BID_1B_FLD_IN_PLACE_SNS,
	BID_2A_FLD_IN_PLACE_SNS,
	BID_2B_FLD_IN_PLACE_SNS,
	BID_3A_FLD_IN_PLACE_SNS,
	BID_3B_FLD_IN_PLACE_SNS,
	BID_4A_FLD_IN_PLACE_SNS,
	BID_4B_FLD_IN_PLACE_SNS,
	BID_5A_FLD_IN_PLACE_SNS,
	BID_5B_FLD_IN_PLACE_SNS,
	BID_6A_FLD_IN_PLACE_SNS,
	BID_6B_FLD_IN_PLACE_SNS,
	RDU_BAK_STROK_SNS,
	RDU_STROK_END_SNS,
	TUBE_ENG_SNS,
	TUBE_DISENG_SNS,
	EXTRCT_PIST_TOP_SNS,
	EXTRCT_ALMST_EMPTY_SNS,
	EXTRCT_PIST_BOTTOM_SNS,
	RDU_PUMP_INLET_PRSR_SNS,
	TUB_SLDR_CLOSE_SNS,
	TUB_SLDR_OPEN_SNS,
	RVLVR_ROTAT_PB,
	RVLVR_UP_SNS,
	RVLVR_DOWN_SNS,
	CD_TNK_LOW_SNS,
	CD_TNK_HI_SNS,
	IDS_TNK_IN_PRSR_SNS,
	IDS_TNK_OUT_PRSR_SNS,
	IDS_BID_TMP_SNS,
	IDS_BID_PRSR_SNS,
	RT_HTR_FLOW_SNS,
	LT_HTR_FLOW_SNS,
	RT_HTR_TMP_SNS,
	LT_HTR_TMP_SNS,
	OFIR_PUMP_ON_IND,
	OFIR_VAC_SWCH,
	OFIR_PRSR_SNS,
	OFIR_VAC_SNS,
	LPH_FOCUS_FRNT_HOME_SNS,
	LPH_FOCUS_RR_HOME_SNS,
	ASID_RUNOUT_FRNT_SNS,
	ASID_RUNOUT_RR_SNS,
	LPHC_TANK_TEMP_SNS,
	LPHC_TANK_LVL_SNS,
	LPHC_PRSR_SNS,
	LPHC_CWS_FLOW_SNS,
	LPHC_LINE_FLOW_SNS,
	LPHC_CWS_TEMP_SNS,
	LPHC_LINE_TEMP_SNS,
	WEB_SPEED,
	IBS_EMPTY_SNS,
	IBS_FULL_SNS,
	RI_MOTOR_HOME_SNS,
	RI_SMPLX_1ST_SNS,
	RI_SMPLX_2ND_SNS,
	IMP_TMP_SNS,
	FI_FRNT_LC,
	FI_RR_LC,
	IBS_FRNT_LC,
	IBS_RR_LC,
	FP_FRNT_LC,
	FP_RR_LC,
	FE_FRNT_LC,
	FE_RR_LC,
	PE_SWF_PB,
	PE_THRD_PB,
	PWS_WG_HOME_SNS,
	PWS_SPLICE_DET_SNS_1,
	PWS_SPLICE_DET_SNS_2,
	IBS_ZONE_TMP_SNS,
	EXT_ZONE_TMP_SNS,
	UW_DIAMETER_SNS,
	UW_DANCER_POS,
	UW_DANCER_TOP_POS,
	UW_DANCER_MID_POS,
	UW_DANCER_BOT_POS,
	UW_BUFF_EMPTY_SNS,
	UW_ROLL_DWN_BTN,
	UW_ROLL_UP_BTN,
	UW_ROLL_IN_TOP_POS,
	UW_TSP_RUN_BTN,
	UW_TSP_STOP_BTN,
	UW_WEB_BRK_SNS,
	RW_DIAMETER_SNS,
	RW_DANCER_POS,
	PACKER_ARM_FDBK,
	RW_DANCER_REG_FDBK,
	SPM_X_POS_HOME_SNS,  
	SPM_Z_POS_HOME_SNS,
	OLS_MTR_HOME_SNS,
	OLS_TRIG_SNS_FEED,
	OLS_TRIG_SNS_EXIT,
	ILP_PRMR_IN_PLACE,
	ILP_CLNR_IN_PLACE,
	ILP_PRMR_ALMST_EMPTY,
	ILP_PRMR_EMPTY,
	ILP_PRMR_FULL,
	ILP_CLNR_ALMST_EMPTY,
	ILP_CLNR_EMPTY,
	ILP_CLNR_FULL,
	ILP_BUFFER_POSITION,
	ILP_DRYER_TEMP_SNS_A,
	ILP_DRYER_TEMP_SNS_B,
	ILP_COR_AIR_SNS_A,
	ILP_COR_AIR_SNS_B,
	ILP_FB_NIP_PB,
	ILP_SWF_PB,
	ILP_WASH_PB,
	IOS_IMO_CLN_HI_LVL_SNS, 
	IOS_IMO_CLN_LO_LVL_SNS, 
	IOS_DIRT_IMO_LVL_SNS,
	IOS_RES_TEMP_SNS,
	ISO_IMO_COND_SNS,
	ISO_IMO_DIRTINESS, 
	IOS_RES_COVER_SNS,
	IOS_DISTILD_TNK_FULL_SNS,
	IOS_SEPRTR_PIPE_FULL_SNS,
	IOS_WTR_LVL_LOW_SNS,
	IOS_CNTRL_FLOW_SNS,
	IOS_CS1_FLOW_METER,
	IOS_CS2_FLOW_METER,
	IOS_CS3_FLOW_METER,
	IOS_CS4_FLOW_METER,
	IOS_CS5_FLOW_METER,
	IOS_CS6_FLOW_METER,
	IOS_CS1_HX_TMP_SNS, 
	IOS_CS2_HX_TMP_SNS, 
	IOS_CS3_HX_TMP_SNS, 
	IOS_CS4_HX_TMP_SNS, 
	IOS_CS5_HX_TMP_SNS, 
	IOS_CS6_HX_TMP_SNS, 
	IOS_CS1_HTR_TMP_SNS,
	IOS_CS2_HTR_TMP_SNS,
	IOS_CS3_HTR_TMP_SNS,
	IOS_CS4_HTR_TMP_SNS,
	IOS_CS5_HTR_TMP_SNS,
	IOS_CS6_HTR_TMP_SNS,
	IOS_INLET_FLTR_PRSSR_SNS,
	IOS_FLTR_A_PRSSR_SNS,
	IOS_FLTR_B_PRSSR_SNS,
	IOS_CS_BFFR_LVL_PRSSR_SNS,
	IOS_CS_RTRN_PUMP_PRSSR_SNS,
	IOS_RIO_BTL_IN_PLAC_SNS, 
	IOS_RIO_BTL_FULL_SNS,
	UC_WST_TRAY_HIGH_LVL_SNS,
	UC_WST_TRAY_LOW_LVL_SNS,
	PE_WST_TRAY_HIGH_LVL_SNS, 
	PE_WST_TRAY_LOW_LVL_SNS,
	EXCES_OIL_PRS_SNS,
	OIL_WST_BTL_IN_PLAC_SNS, 
	OIL_WST_BTL_FULL_SNS,
	CVC1_A_IN_TMP_SNS,
	CVC1_B_IN_TMP_SNS,
	CVC2_A_IN_TMP_SNS,
	CVC2_B_IN_TMP_SNS,
	CVC1_AIR_ECO_PRS_SNS,
	CVC2_AIR_ECO_PRS_SNS,
	CVC1_WTR_ECO_FLOW,
	CVC2_WTR_ECO_FLOW,
	CVC1_WTR_HX_FLOW,
	CVC2_WTR_HX_FLOW,
	CVC1_A_DP_TMP_SNS,
	CVC1_B_DP_TMP_SNS,
	CVC2_A_DP_TMP_SNS,
	CVC2_B_DP_TMP_SNS,
	CVC1_A_OUT_TMP_SNS,
	CVC1_B_OUT_TMP_SNS,
	CVC2_A_OUT_TMP_SNS,
	CVC2_B_OUT_TMP_SNS,
	CVC1_AIR_OUT_PRS_SNS,
	CVC2_AIR_OUT_PRS_SNS,
	CVC1_A_BLWR_PRS_SNS,
	CVC1_B_BLWR_PRS_SNS,
	CVC2_A_BLWR_PRS_SNS,
	CVC2_B_BLWR_PRS_SNS,
	CVC1_A_BLWR_SPD_ERR,
	CVC1_B_BLWR_SPD_ERR,
	CVC2_A_BLWR_SPD_ERR,
	CVC2_B_BLWR_SPD_ERR,
	CVC1_A_BLWR_SPD_IND,
	CVC1_B_BLWR_SPD_IND,
	CVC2_A_BLWR_SPD_IND,
	CVC2_B_BLWR_SPD_IND,
	CVC_TNK_LVL_SNS,
	CVC_PMP_PRS_SNS,
	MTC_1_SNS,
	MTC_2_SNS,
	MTC_3_SNS,
	MTC_4_SNS,
	MHC_1_SNS,
	MHC_2_SNS,
	MHC_3_SNS,
	MHC_4_SNS,
	CWS_PRE_FLTR_PRSR,
	CWS_POST_FLTR_PRSR,
	CWS_TEMP_SNSR, 
	CWS_FLOW_SENSOR,
	CWS_CHILLER_ALRM,
	CWS_CHILLER_CNTR,
	FEED_EC_FAN1_FDBK,
	FEED_EC_FAN2_FDBK,
	FEED_EC_FAN3_FDBK,
	EXIT_EC_FAN1_FDBK,
	EXIT_EC_FAN2_FDBK,
	EXIT_EC_FAN3_FDBK,
	EC_AMBIENT_TMP,
	UC_EC_FANS_FDBK,
	UC_PNMTK_PRSR_SNS,
	FRNT_DOOR_INTLK,
	PE_FRNT_DOOR_INTLK,
	PE_FRNT_DOOR_OPN_REQ,
	PE_THRD_FEED_DOOR_INTLK,
	PE_FRNT_THRD_EXIT_DOOR_INTLK,
	PE_RR_FEED_DOOR_INTLK,
	PE_RR_EXIT_DOOR_INTLK,
	PE_RR_EXIT_DOOR_OPN_REQ,
	PWS_FRNT_FEED_DOOR_INTLK,
	PWS_FRNT_FEED_DOOR_OPN_REQ,
	PWS_FRNT_EXIT_DOOR_INTLK,
	PWS_RR_EXIT_DOOR_INTLK,
	PWS_RR_EXIT_DOOR_OPN_REQ,
	UIC_THRD_FEED_DOOR_INTLK,
	UIC_THRD_EXIT_DOOR_INTLK,
	EFS_1_INTRLK,
	EFS_2_INTRLK,
	PE_FRNT_EMS,
	PE_RR_EMS,
	PWS_FRNT_EMS,
	PWS_RR_EMS,
	UIC_FRNT_FEED_EMS,
	UIC_FRNT_EXIT_EMS,
	UIC_RR_EMS,
	UIC_OPER_EMS,
	UW_EMS,
	RW_EMS
)DINT;
END_TYPE

// ---- DUTs/Motion/Enums/eStationNo.TcDUT
{attribute 'qualified_only'}
//{attribute 'strict'}
{attribute 'to_string'}
TYPE eStationNo :
(
	Station1 := 1,
	Station2 := 2,
	Station3 := 3,
	Station4 := 4,
	Station5 := 5,
	Station6 := 6,
	Station7 := 7
)DINT;
END_TYPE

// ---- DUTs/Motion/Enums/eSubsystemID.TcDUT
{attribute 'qualified_only'}
//{attribute 'strict'}
{attribute 'to_string'}
TYPE eSubsystemID :
(
	NoSubsystem := 0,
	General ,
	Safety ,
	Blanket ,
	Station_1 ,
	Station_2 ,
	Station_3 ,
	Station_4 ,
	Station_5 ,
	Station_6 ,
	WHS ,
	ILP	,
	ImagingOil ,
	AmbientControl ,
	ELC ,
	ITM	,
	BKT_Tension	,
	BKT_Centering ,
	BR_St_1	,
	BR_St_2	,
	BR_St_3 ,
	BR_St_4	,
	BR_St_5	,
	BR_St_6	,
	BKT_Drying,
	BKT_HeatElement_1 ,
	BKT_HeatElement_2 ,
	BKT_HeatElement_3 ,
	BKT_HeatElement_4 ,
	BKT_HeatElement_5 ,
	BKT_HeatElement_6 ,
	BKT_HeatElement_7 ,
	BKT_HeatElement_8 ,
	BKT_HeatElement_9 ,
	BKT_HeatElement_10 ,
	BRU	,
	Asid_Stn_1 ,
	Asid_Stn_2 ,
	Asid_Stn_3 ,
	Asid_Stn_4 ,
	Asid_Stn_5 ,
	Asid_Stn_6 ,
	LPH_Stn_1 ,
	LPH_Stn_2 ,
	LPH_Stn_3 ,
	LPH_Stn_4 ,
	LPH_Stn_5 ,
	LPH_Stn_6 ,
	LPH_Cooling ,
	CS_Stn_1 ,
	CS_Stn_2 ,
	CS_Stn_3,
	CS_Stn_4 ,
	CS_Stn_5 ,
	CS_Stn_6 ,
	BID_Manager_1_Stn_1 ,
	BID_Manager_2_Stn_1 ,
	BID_Manager_1_Stn_2 ,
	BID_Manager_2_Stn_2 ,
	BID_Manager_1_Stn_3 ,
	BID_Manager_2_Stn_3 ,
	BID_Manager_1_Stn_4 ,
	BID_Manager_2_Stn_4 ,
	BID_Manager_1_Stn_5 ,
	BID_Manager_2_Stn_5 ,
	BID_Manager_1_Stn_6 ,
	BID_Manager_2_Stn_6 ,
	BID_Rot_1_Stn_1 ,
	BID_Rot_2_Stn_1	,
	BID_Rot_1_Stn_2	,
	BID_Rot_2_Stn_2	,
	BID_Rot_1_Stn_3	,
	BID_Rot_2_Stn_3	,
	BID_Rot_1_Stn_4	,
	BID_Rot_2_Stn_4 ,
	BID_Rot_1_Stn_5	,
	BID_Rot_2_Stn_5	,
	BID_Rot_1_Stn_6	,
	BID_Rot_2_Stn_6	,
	BID_Eng_1_Stn_1	,
	BID_Eng_2_Stn_1	,
	BID_Eng_1_Stn_2	,
	BID_Eng_2_Stn_2	,
	BID_Eng_1_Stn_3	,
	BID_Eng_2_Stn_3	,
	BID_Eng_1_Stn_4	,
	BID_Eng_2_Stn_4 ,
	BID_Eng_1_Stn_5	,
	BID_Eng_2_Stn_5	,
	BID_Eng_1_Stn_6	,
	BID_Eng_2_Stn_6	,
	BID_HV_1_Stn_1 ,
	BID_HV_2_Stn_1 ,
	BID_HV_1_Stn_2 ,
	BID_HV_2_Stn_2 ,
	BID_HV_1_Stn_3 ,
	BID_HV_2_Stn_3 ,
	BID_HV_1_Stn_4 ,
	BID_HV_2_Stn_4 ,
	BID_HV_1_Stn_5 ,
	BID_HV_2_Stn_5 ,
	BID_HV_1_Stn_6 ,
	BID_HV_2_Stn_6 ,
	INK_1_Stn_1	,
	INK_2_Stn_1	,
	INK_1_Stn_2	,
	INK_2_Stn_2 ,
	INK_1_Stn_3	,
	INK_2_Stn_3	,
	INK_1_Stn_4	,
	INK_2_Stn_4	,
	INK_1_Stn_5	,
	INK_2_Stn_5	,
	INK_1_Stn_6	,
	INK_2_Stn_6	,
	AsidChargeHV_Stn_1 ,
	AsidChargeHV_Stn_2 ,
	AsidChargeHV_Stn_3 ,
	AsidChargeHV_Stn_4 ,
	AsidChargeHV_Stn_5 ,
	AsidChargeHV_Stn_6 ,
	CR_Engage_Stn_1 ,
	CR_Engage_Stn_2 ,
	CR_Engage_Stn_3 ,
	CR_Engage_Stn_4 ,
	CR_Engage_Stn_5 ,
	CR_Engage_Stn_6 ,
	InkWater_1 ,
	InkWater_2 ,
	UW ,
	WHS_Internal ,
	WHS_Impression ,
	WHS_Buffer ,
	SPM ,
	RW ,
	Primer ,
	Dryer ,
	Corona ,
	IMO_Reservoir ,
	IMO_Recycle ,
	IMO_Waste ,
	IMO_Temperature ,
	IMO_Flow ,
	IMO_Dirtiness ,
	ITC ,
	CWS ,
	CVC ,
	Manager,
	LAST 
)DINT;
END_TYPE

// ---- DUTs/Motion/Enums/eVendorNameID.TcDUT
{attribute 'qualified_only'}
//{attribute 'strict'}
{attribute 'to_string'}
TYPE eVendorNameID :
(	
	NoVendor := 		0,
	BR := 				1,
	Beckhoff := 		2,
	Elmo := 			3,
	ControlTechnique :=	4,
	Servotronics := 	5,
	Nidec :=			6,
	LAST		
)DINT;
END_TYPE

// ---- DUTs/Motion/ExtendedAxisTyp.TcDUT
TYPE ExtendedAxisTyp  :
	STRUCT
		Basic_axis 	: Basic_axis_typ;
		MultiAxis 	: MultiAxis_typ;
		CyclicAxis	: CyclicAxis_typ;
		ParIDAccess	: ParIDAccess_Typ;
		VelocityCtrl: VelocityCtrl_typ;
	END_STRUCT
END_TYPE

// ---- DUTs/Motion/STRUCT_AxisExtendedCompound.TcDUT
TYPE STRUCT_AxisExtendedCompound :
STRUCT
	
	Ref:		AXIS_REF;
	Crtl:		ExtendedAxisTyp;
	
END_STRUCT
END_TYPE

// ---- DUTs/Motion/WebAxes_typ.TcDUT
TYPE WebAxes_typ :
STRUCT
	
	// Winding	
	UwVmaster	: 	STRUCT_AxisExtendedCompound;
	UW_1		:  STRUCT_AxisExtendedCompound;
	UW_2		:  STRUCT_AxisExtendedCompound;	
	Output		:  STRUCT_AxisExtendedCompound;
	
END_STRUCT
END_TYPE

// ---- DUTs/Motion/Winders/DancerTyp.TcDUT
TYPE DancerTyp :
STRUCT
	stLutDataParam				:ST_LookUpTableParam;
	DancerPosition_Unfiltred	:LREAL;
	DancerLPF					:FB_LPF;
	DancerPosition_filtred		:LREAL;	
	fb_DancerCtrl				:FB_DancerCtrl;
	
	DancerGear:LREAL;
END_STRUCT
END_TYPE

// ---- DUTs/Motion/Winders/Dimeter_Typ.TcDUT
TYPE Dimeter_Typ :
STRUCT
	
	stLutDataParam:	ST_LookUpTableParam;
	Diameter_Unfiltred	:LREAL;
	DiameterLPF:			FB_LPF;
	Diameter_filtred	:LREAL;
	

END_STRUCT
END_TYPE

// ---- DUTs/Motion/Winders/E_DancerCtrlTyp.TcDUT
//{attribute 'qualified_only'}
//{attribute 'strict'}
TYPE E_DancerCtrlTyp :
(
	DIGITAL := 0,
	ANALOG	:=10
);
END_TYPE

// ---- DUTs/Motion/Winders/Tension_Typ.TcDUT
TYPE Tension_Typ :
STRUCT
	stLutDataParam		:ST_LookUpTableParam;
	Tension_Unfiltred	:LREAL;
	LoadCellLPF			:FB_LPF;
	Tension_filtred		:LREAL;
	FB_TensionLoop:FB_TensionLoop;
	
	TensionGear:LREAL;
END_STRUCT
END_TYPE

// ---- DUTs/Motion/Winders/WinderParam_Typ.TcDUT
TYPE WinderParam_Typ :
STRUCT
	
	CalculatedRotSpeed:LREAL;
	CalculatedGear:LREAL;
	Tension:Tension_Typ;
	Dancer:DancerTyp;
END_STRUCT
END_TYPE

// ---- POUs/Lib/CH Obj/CH_Typ/Basic_cycle_CMD_typ.TcDUT
TYPE Basic_cycle_CMD_typ :
	STRUCT
		Start 						: BOOL; (* cycle start*)
		Pause 						: BOOL; (*cycle pause*)
		ResetErr 					: BOOL; (*reset cycle fault*)
		Resume 						: BOOL; (*resume after Pause*)
		ResetCycle 					: BOOL; (*Cycle reset*)
		StepByStep 					: BOOL; (* operate the cycle step by step *)
		SetFaultEvent				: BOOL;  // Triggers Fault Event 
		DeactivateStepTimeOut 		: BOOL; (*If Input is On Process will Not Go to TimeOut Fault*) (* From Function *)
		Deacivate_Sequence_Time_Out : BOOL;
		LogMsgInit 					: BOOL := TRUE;
		EnableStateLogging			: BOOL;
		WriteExternalFaultLogCMD	: BOOL;
		WriteExternalLogCMD			: BOOL;
	END_STRUCT
END_TYPE

// ---- POUs/Lib/CH Obj/CH_Typ/Basic_cycle_Input.TcDUT
TYPE Basic_cycle_Input :
	STRUCT
		CMD 		: Basic_cycle_CMD_typ;
		Parameter 	: Basic_cycle_Param_typ;
		Delay 		: TON;
	END_STRUCT
END_TYPE

// ---- POUs/Lib/CH Obj/CH_Typ/Basic_cycle_Mon_typ.TcDUT
TYPE Basic_cycle_Mon_typ :
	STRUCT
		StepNo 				: DINT; (* current cycle step *)
		PrevStepNo 			: DINT; (* previous cycle step *)
		SubStepNo 			: DINT; (* current cycle step *)
		StepMessage 		: STRING[100]; (* Inside the Cycle *)
		SubStepMessage 		: STRING[100]; (* Inside the Cycle *)
		LastStep 			: DINT;
		Error_Text 			: STRING[100];
		External_Error_Text : STRING[100];
		Visu_StepNo 		: DINT;
		LastCycleTime 		: TIME;
		CycleTime 			: TIME;
		Step_TimeOut 		: TIME;
		SubStep_TimeOut 	: TIME;
		ExternalLogText		: STRING[100];
		ExternalLogParam1	: DINT;
		
	END_STRUCT
END_TYPE

// ---- POUs/Lib/CH Obj/CH_Typ/Basic_cycle_Output.TcDUT
TYPE Basic_cycle_Output :
	STRUCT
		Status 	: Basic_cycle_Status_typ;
		Monitor : Basic_cycle_Mon_typ;
		Error 	: Error_Handler_typ;
	END_STRUCT
END_TYPE

// ---- POUs/Lib/CH Obj/CH_Typ/Basic_cycle_Param_typ.TcDUT
TYPE Basic_cycle_Param_typ :
	STRUCT
		TimeOut 		: TIME;
		CycleTimeOut 	: TIME;
		ThreadName 		: STRING[50];
		CHName 			: STRING[20];
		PosForLog 		: USINT;
		StepMessageIsForNewState	: BOOL := FALSE; (* indicate that StepMessage is set for StepNo that be moving to; is FALSEd right after printing the log *)
		ExternalLogType :enumLogMessageLevelSeverity ;
		
	END_STRUCT
END_TYPE

// ---- POUs/Lib/CH Obj/CH_Typ/Basic_cycle_Status_typ.TcDUT
TYPE Basic_cycle_Status_typ :
	STRUCT
		CycleTimeOut_Fault 	: BOOL;
		Running 			: BOOL; (*cycle is  running*)
		Fault 				: BOOL; (*cycle at fault*)
		Done 				: BOOL; (* cycle Done *)
		CycleStuck 			: BOOL;
		SubStepStuck 		: BOOL ;
	END_STRUCT
END_TYPE

// ---- POUs/Lib/CH Obj/CH_Typ/Basic_cycle_typ.TcDUT
TYPE Basic_cycle_typ :
	STRUCT
		Input 	: Basic_cycle_Input;
		Output 	: Basic_cycle_Output;
	END_STRUCT
END_TYPE

// ---- POUs/Lib/CH Obj/CH_Typ/CH_ErrorReport_typ.TcDUT
TYPE CH_ErrorReport_typ :
	STRUCT
		MessageID 			: DINT;
		FailureType 		: DINT;
		FailureSubType 		: DINT;
		FailedUnitID 		: DINT;
		Severity 			: DINT;
		ErrorCode 			: DINT;
		AlarmID 			: UINT;
		SheetID 			: UDINT;
		RefID 				: UDINT;
		ActualValue 		: UINT;
		ViolatedThreshold 	: UINT;
	END_STRUCT
END_TYPE

// ---- POUs/Lib/CH Obj/CH_Typ/Error_Handler_typ.TcDUT
TYPE Error_Handler_typ :
	STRUCT
		//ErrorHandler 	: ERR_HANDLER_typ;
		//ErrorInfo 	: ERR_TASK_INFO_typ;
	END_STRUCT
END_TYPE

// ---- POUs/Lib/Events/Enums/eMotorID_1.TcDUT
{attribute 'qualified_only'}
//{attribute 'strict'}
{attribute 'to_string'}
TYPE eMotorID_1 :
(
	NoMotor := 	0,
	ITM ,
	BKT_TensionFront ,
	BKT_TensionRear ,
	BKT_LateralFront ,
	BKT_LateralRear ,
	BKT_HeaterLowerAirKnivesBlower ,
	BKT_HeaterUpperAirKnivesBlower ,
	BlanketEngageFrontValve_1 ,
	BlanketEngageFrontValve_2 ,
	BlanketEngageFrontValve_3 ,
	BlanketEngageFrontValve_4 ,
	BlanketEngageFrontValve_5 ,
	BlanketEngageFrontValve_6 ,
	BlanketEngageRearValve_1 ,
	BlanketEngageRearValve_2 ,
	BlanketEngageRearValve_3 ,
	BlanketEngageRearValve_4 ,
	BlanketEngageRearValve_5 ,
	BlanketEngageRearValve_6 ,
	BKT_FeedSupportRoller ,
	BKT_EdgeSensorFan ,
	BKT_IndexSensorFan ,
	BKT_RegCamerasCoolingValve ,
	BRU_StickyRotate ,
	BRU_StickyEngageFront ,
	BRU_StickyEngageRear ,
	BRU_Heater ,
	BRU_StickyPeeling ,
	BRU_StickyServiceDisengage ,
	BRU_BWS ,
	BWS_MiteringPump ,
	BWS_CirculationPump ,	
	ASID_Drive ,
	ChargeRollerEngage ,
	LPH_EngageFront ,
	LPH_EngageRear ,
	LPH_CoolingValve ,
	LPH_CoolingPump ,
	LPH_CoolingTankHeater ,
	CS_WettingRoller ,
	CS_CollectingRoller ,
	CS_Engage ,
	CS_Disengage ,
	CR_Engage ,
	BID_Drive ,
	BID_EngageFront ,
	BID_EngageRear ,
	INK_ChargeDirectorPump ,
	INK_to_BID_pump ,
	INK_RDU_Valve ,
	INK_ExtractionPistonDown ,
	INK_ExtractionPistonUp ,
	INK_TubeEngageValve ,
	INK_TubeDisengageValve ,
	INK_TubeSliderPiston ,
	INK_RevolverLiftValve ,
	UW_Roller ,
	UW_ArmsUp ,
	UW_ArmsDown ,
	UW_RightClamp ,
	UW_LeftClamp ,
	UW_WebGuide ,
	WHS_FI ,
	WHS_PTR ,
	WHS_IPE_Front ,
	WHS_IPE_Rear ,
	WHS_IMP ,
	WHS_Peeler ,
	WHS_FP ,
	WHS_FE ,
	WHS_FI_NipEngageValve ,
	WHS_FI_NipDisengageValve ,
	WHS_FR_NipValve ,
	WHS_FP_NipEngageValve ,
	WHS_FP_NipDisengageValve ,
	WHS_FE_NipEngageValve ,
	WHS_FE_NipDisengageValve ,
	WHS_PE_WebGuide ,
	WHS_IBS ,
	WHS_BRI ,
	WHS_BRO ,
	WHS_ReinsertionXposition  ,
	RW_Roller ,
	RW_RightClamp,
	RW_LeftClamp ,
	RW_AirShaft ,
	RW_PackerArm  ,
	SPM_X ,
	SPM_Z ,
	ILP_FI_Motor ,
	ILP_FI_Nip ,
	ILP_FB_Motor ,
	ILP_FB_NipEngage ,
	PrimingMotor ,
	PrimingPump ,
	PrimerInputValve ,
	PrimerOutputValve ,
	DrainValve ,
	LowerRubberRollerEngage ,
	UpperRubberRollerEngage ,
	ImpressionEngage ,
	ILP_DryerBlower ,
	ILP_DryerExhaust ,
	ILP_DryerHeater ,
	ILP_FastCoolingValve ,
	ILP_CORONA_Ozone_Suction ,
	CVC1A_CoolingBlower ,
	CVC1B_CoolingBlower ,
	CVC2A_CoolingBlower ,
	CVC2B_CoolingBlower ,
	CVC_WaterPump ,
	CVC_WaterSupply  ,
	CVC_WaterReturn ,
	CVC_HX_WaterValve ,
	IMO_CS_CoolingHigh_1 ,
	IMO_CS_CoolingHigh_2 ,
	IMO_CS_CoolingHigh_3 ,
	IMO_CS_CoolingHigh_4 ,
	IMO_CS_CoolingHigh_5 ,
	IMO_CS_CoolingHigh_6 ,
	IMO_CS_CoolingMid_1 ,
	IMO_CS_CoolingMid_2 ,
	IMO_CS_CoolingMid_3 ,
	IMO_CS_CoolingMid_4 ,
	IMO_CS_CoolingMid_5 ,
	IMO_CS_CoolingMid_6 ,
	IMO_CS_CoolingLow_1 ,
	IMO_CS_CoolingLow_2 ,
	IMO_CS_CoolingLow_3 ,
	IMO_CS_CoolingLow_4 ,
	IMO_CS_CoolingLow_5 ,
	IMO_CS_CoolingLow_6 ,
	IMO_CS_InletPump_1 ,
	IMO_CS_InletPump_2 ,
	IMO_CS_InletPump_3 ,
	IMO_CS_InletPump_4 ,
	IMO_CS_InletPump_5 ,
	IMO_CS_InletPump_6 ,
	IMO_CS_ReturnPump ,
	IMO_EFS_Motor ,
	IMO_EFS_FilterPump ,
	IMO_PE_WastePump ,
	IMO_UC_WastePump ,
	IWS_WaterPumpRight,
	IWS_WaterPumpLeft,
	IWS_InputValveRight,	
	IWS_InputValveLeft,	
	IWS_InkWaterValve_1,	
	IWS_InkWaterValve_2,	
	IWS_InkWaterValve_3,	
	IWS_InkWaterValve_4,	
	IWS_InkWaterValve_5,	
	IWS_InkWaterValve_6,	
	IWS_InkWaterValve_7,	
	IWS_InkWaterValve_8,	
	IWS_InkWaterValve_9,	
	IWS_InkWaterValve_10,	
	IWS_InkWaterValve_11,	
	IWS_InkWaterValve_12,	
	UC_EC_Fans_1 ,
	UC_EC_Fans_2 ,
	UC_EC_Fans_3 ,
	UC_EC_Fans_4 ,
	LAST 
)DINT;
END_TYPE

// ---- POUs/Lib/Events/Enums/eSensorID_1.TcDUT
{attribute 'qualified_only'}
//{attribute 'strict'}
{attribute 'to_string'}
TYPE eSensorID_1 :
(
	NoSensor,
	BKT_EDGE_SNS,
	BKT_IND_NPN_SNS,
	BKT_IND_PNP_SNS, 
	BKT_TENS_FRNT_HOME_SNS, 
	BKT_TENS_RR_HOME_SNS,
	BKT_TENS_FRNT_LD_CELL,
	BKT_TENS_RR_LD_CELL,
	BKT_TENS_SAFE_DETCT,
	BKT_LTRL_FRNT_HOME_SNS,
	BKT_LTRL_RR_HOME_SNS,
	SUP_ROLL_HOME_SNS,
	BRU_STKY_PEEL_HOME_SNS,
	BRU_STKY_MID_ROLLER_SNS,
	BRU_STKY_STIR_IN_PLC_SNS,
	BRU_STKY_TRAY_LVL_MID,
	BRU_STKY_TRAY_LVL_TOP,
	BRU_STKY_MID_ROL_TEMP,
	BRU_BWS_IN_PLC_SNS,
	BRU_BWS_FRNT_LIMT_SNS,
	BRU_BWS_RR_LIMT_SNS,
	BRU_BWS_LVL_SW_TOP,
	BRU_BWS_LVL_SW_BOT,
	BRT_SRV_POS_FRNT_1,
	BRT_SRV_POS_FRNT_2,
	BRT_SRV_POS_FRNT_3,
	BRT_SRV_POS_FRNT_4,
	BRT_SRV_POS_FRNT_5,
	BRT_SRV_POS_FRNT_6,
	BRT_SRV_POS_RR_1,
	BRT_SRV_POS_RR_2,
	BRT_SRV_POS_RR_3,
	BRT_SRV_POS_RR_4,
	BRT_SRV_POS_RR_5,
	BRT_SRV_POS_RR_6,
	EH_TMP_SNS_01,
	EH_TMP_SNS_02,
	EH_TMP_SNS_03,
	EH_TMP_SNS_04,
	EH_TMP_SNS_05,
	EH_TMP_SNS_06,
	EH_TMP_SNS_07A,
	EH_TMP_SNS_07B,
	EH_TMP_SNS_08,
	EH_TMP_SNS_09,
	EH_TMP_SNS_10A,
	EH_TMP_SNS_10B,
	EH_HOOD_IN_PLC_SNS_07,
	EH_HOOD_IN_PLC_SNS_08,
	EH_HOOD_IN_PLC_SNS_09,
	EH_HOOD_IN_PLC_SNS_10,
	EH_SUC_PRSSR_SNS_01,
	EH_SUC_PRSSR_SNS_02,
	EH_SUC_PRSSR_SNS_03,
	EH_SUC_PRSSR_SNS_04,
	EH_SUC_PRSSR_SNS_05,
	EH_SUC_PRSSR_SNS_06,
	EH_SUC_PRSSR_SNS_07,
	EH_SUC_PRSSR_SNS_08,
	EH_SUC_PRSSR_SNS_09,
	EH_SUC_PRSSR_SNS_10,
	EH_TOP_AIR_KNF_PRSSR_SNS,
	EH_BTM_AIR_KNF_PRSSR_SNS,
	EH_TOP_AIR_KNF_BLWR_TMP,
	EH_BTM_AIR_KNF_BLWR_TMP,
	EH_AIR_PRG_PRSSR_SNS,
	ITM_DRUM_FRNT_TEMP_SNS, 
	ITM_DRUM_RR_TEMP_SNS,
	EBV_SUC_PRS_SNS,
	EBV_TEMP_SNS,
	ITC_TMP_SNS,
	ITC_LVL_SNS,
	ASID_IN_PLC_SNS,
	ASID_DRUM_TEMP_SNS,
	ASID_DRV_TEMP,
	CR_IN_PLC_SNS,
	CR_DISENG_FRT_SNS,
	CR_DISENG_RR_SNS,
	ELECTROMETER_OUT,
	CS_IN_PLC_SNS,
	CS_ENG_SNS,
	CS_DISENG_SNS,
	CS_AIR_PRSR_SNS,
	CS_TEMP_SNS,
	BID_1A_FLD_IN_PLACE_SNS,
	BID_1B_FLD_IN_PLACE_SNS,
	BID_2A_FLD_IN_PLACE_SNS,
	BID_2B_FLD_IN_PLACE_SNS,
	BID_3A_FLD_IN_PLACE_SNS,
	BID_3B_FLD_IN_PLACE_SNS,
	BID_4A_FLD_IN_PLACE_SNS,
	BID_4B_FLD_IN_PLACE_SNS,
	BID_5A_FLD_IN_PLACE_SNS,
	BID_5B_FLD_IN_PLACE_SNS,
	BID_6A_FLD_IN_PLACE_SNS,
	BID_6B_FLD_IN_PLACE_SNS,
	RDU_BAK_STROK_SNS,
	RDU_STROK_END_SNS,
	TUBE_ENG_SNS,
	TUBE_DISENG_SNS,
	EXTRCT_PIST_TOP_SNS,
	EXTRCT_ALMST_EMPTY_SNS,
	EXTRCT_PIST_BOTTOM_SNS,
	RDU_PUMP_INLET_PRSR_SNS,
	TUB_SLDR_CLOSE_SNS,
	TUB_SLDR_OPEN_SNS,
	RVLVR_ROTAT_PB,
	RVLVR_UP_SNS,
	RVLVR_DOWN_SNS,
	CD_TNK_LOW_SNS,
	CD_TNK_HI_SNS,
	IDS_TNK_IN_PRSR_SNS,
	IDS_TNK_OUT_PRSR_SNS,
	IDS_BID_TMP_SNS,
	IDS_BID_PRSR_SNS,
	RT_HTR_FLOW_SNS,
	LT_HTR_FLOW_SNS,
	RT_HTR_TMP_SNS,
	LT_HTR_TMP_SNS,
	OFIR_PUMP_ON_IND,
	OFIR_VAC_SWCH,
	OFIR_PRSR_SNS,
	OFIR_VAC_SNS,
	LPH_FOCUS_FRNT_HOME_SNS,
	LPH_FOCUS_RR_HOME_SNS,
	ASID_RUNOUT_FRNT_SNS,
	ASID_RUNOUT_RR_SNS,
	LPHC_TANK_TEMP_SNS,
	LPHC_TANK_LVL_SNS,
	LPHC_PRSR_SNS,
	LPHC_CWS_FLOW_SNS,
	LPHC_LINE_FLOW_SNS,
	LPHC_CWS_TEMP_SNS,
	LPHC_LINE_TEMP_SNS,
	WEB_SPEED,
	IBS_EMPTY_SNS,
	IBS_FULL_SNS,
	RI_MOTOR_HOME_SNS,
	RI_SMPLX_1ST_SNS,
	RI_SMPLX_2ND_SNS,
	IMP_TMP_SNS,
	FI_FRNT_LC,
	FI_RR_LC,
	IBS_FRNT_LC,
	IBS_RR_LC,
	FP_FRNT_LC,
	FP_RR_LC,
	FE_FRNT_LC,
	FE_RR_LC,
	PE_SWF_PB,
	PE_THRD_PB,
	PWS_WG_HOME_SNS,
	PWS_SPLICE_DET_SNS_1,
	PWS_SPLICE_DET_SNS_2,
	IBS_ZONE_TMP_SNS,
	EXT_ZONE_TMP_SNS,
	UW_DIAMETER_SNS,
	UW_DANCER_POS,
	UW_DANCER_TOP_POS,
	UW_DANCER_MID_POS,
	UW_DANCER_BOT_POS,
	UW_BUFF_EMPTY_SNS,
	UW_ROLL_DWN_BTN,
	UW_ROLL_UP_BTN,
	UW_ROLL_IN_TOP_POS,
	UW_TSP_RUN_BTN,
	UW_TSP_STOP_BTN,
	UW_WEB_BRK_SNS,
	RW_DIAMETER_SNS,
	RW_DANCER_POS,
	PACKER_ARM_FDBK,
	RW_DANCER_REG_FDBK,
	SPM_X_POS_HOME_SNS,  
	SPM_Z_POS_HOME_SNS,
	OLS_MTR_HOME_SNS,
	OLS_TRIG_SNS_FEED,
	OLS_TRIG_SNS_EXIT,
	ILP_PRMR_IN_PLACE,
	ILP_CLNR_IN_PLACE,
	ILP_PRMR_ALMST_EMPTY,
	ILP_PRMR_EMPTY,
	ILP_PRMR_FULL,
	ILP_CLNR_ALMST_EMPTY,
	ILP_CLNR_EMPTY,
	ILP_CLNR_FULL,
	ILP_BUFFER_POSITION,
	ILP_DRYER_TEMP_SNS_A,
	ILP_DRYER_TEMP_SNS_B,
	ILP_COR_AIR_SNS_A,
	ILP_COR_AIR_SNS_B,
	ILP_FB_NIP_PB,
	ILP_SWF_PB,
	ILP_WASH_PB,
	IOS_IMO_CLN_HI_LVL_SNS, 
	IOS_IMO_CLN_LO_LVL_SNS, 
	IOS_DIRT_IMO_LVL_SNS,
	IOS_RES_TEMP_SNS,
	ISO_IMO_COND_SNS,
	ISO_IMO_DIRTINESS, 
	IOS_RES_COVER_SNS,
	IOS_DISTILD_TNK_FULL_SNS,
	IOS_SEPRTR_PIPE_FULL_SNS,
	IOS_WTR_LVL_LOW_SNS,
	IOS_CNTRL_FLOW_SNS,
	IOS_CS1_FLOW_METER,
	IOS_CS2_FLOW_METER,
	IOS_CS3_FLOW_METER,
	IOS_CS4_FLOW_METER,
	IOS_CS5_FLOW_METER,
	IOS_CS6_FLOW_METER,
	IOS_CS1_HX_TMP_SNS, 
	IOS_CS2_HX_TMP_SNS, 
	IOS_CS3_HX_TMP_SNS, 
	IOS_CS4_HX_TMP_SNS, 
	IOS_CS5_HX_TMP_SNS, 
	IOS_CS6_HX_TMP_SNS, 
	IOS_CS1_HTR_TMP_SNS,
	IOS_CS2_HTR_TMP_SNS,
	IOS_CS3_HTR_TMP_SNS,
	IOS_CS4_HTR_TMP_SNS,
	IOS_CS5_HTR_TMP_SNS,
	IOS_CS6_HTR_TMP_SNS,
	IOS_INLET_FLTR_PRSSR_SNS,
	IOS_FLTR_A_PRSSR_SNS,
	IOS_FLTR_B_PRSSR_SNS,
	IOS_CS_BFFR_LVL_PRSSR_SNS,
	IOS_CS_RTRN_PUMP_PRSSR_SNS,
	IOS_RIO_BTL_IN_PLAC_SNS, 
	IOS_RIO_BTL_FULL_SNS,
	UC_WST_TRAY_HIGH_LVL_SNS,
	UC_WST_TRAY_LOW_LVL_SNS,
	PE_WST_TRAY_HIGH_LVL_SNS, 
	PE_WST_TRAY_LOW_LVL_SNS,
	EXCES_OIL_PRS_SNS,
	OIL_WST_BTL_IN_PLAC_SNS, 
	OIL_WST_BTL_FULL_SNS,
	CVC1_A_IN_TMP_SNS,
	CVC1_B_IN_TMP_SNS,
	CVC2_A_IN_TMP_SNS,
	CVC2_B_IN_TMP_SNS,
	CVC1_AIR_ECO_PRS_SNS,
	CVC2_AIR_ECO_PRS_SNS,
	CVC1_WTR_ECO_FLOW,
	CVC2_WTR_ECO_FLOW,
	CVC1_WTR_HX_FLOW,
	CVC2_WTR_HX_FLOW,
	CVC1_A_DP_TMP_SNS,
	CVC1_B_DP_TMP_SNS,
	CVC2_A_DP_TMP_SNS,
	CVC2_B_DP_TMP_SNS,
	CVC1_A_OUT_TMP_SNS,
	CVC1_B_OUT_TMP_SNS,
	CVC2_A_OUT_TMP_SNS,
	CVC2_B_OUT_TMP_SNS,
	CVC1_AIR_OUT_PRS_SNS,
	CVC2_AIR_OUT_PRS_SNS,
	CVC1_A_BLWR_PRS_SNS,
	CVC1_B_BLWR_PRS_SNS,
	CVC2_A_BLWR_PRS_SNS,
	CVC2_B_BLWR_PRS_SNS,
	CVC1_A_BLWR_SPD_ERR,
	CVC1_B_BLWR_SPD_ERR,
	CVC2_A_BLWR_SPD_ERR,
	CVC2_B_BLWR_SPD_ERR,
	CVC1_A_BLWR_SPD_IND,
	CVC1_B_BLWR_SPD_IND,
	CVC2_A_BLWR_SPD_IND,
	CVC2_B_BLWR_SPD_IND,
	CVC_TNK_LVL_SNS,
	CVC_PMP_PRS_SNS,
	MTC_1_SNS,
	MTC_2_SNS,
	MTC_3_SNS,
	MTC_4_SNS,
	MHC_1_SNS,
	MHC_2_SNS,
	MHC_3_SNS,
	MHC_4_SNS,
	CWS_PRE_FLTR_PRSR,
	CWS_POST_FLTR_PRSR,
	CWS_TEMP_SNSR, 
	CWS_FLOW_SENSOR,
	CWS_CHILLER_ALRM,
	CWS_CHILLER_CNTR,
	FEED_EC_FAN1_FDBK,
	FEED_EC_FAN2_FDBK,
	FEED_EC_FAN3_FDBK,
	EXIT_EC_FAN1_FDBK,
	EXIT_EC_FAN2_FDBK,
	EXIT_EC_FAN3_FDBK,
	EC_AMBIENT_TMP,
	UC_EC_FANS_FDBK,
	UC_PNMTK_PRSR_SNS,
	FRNT_DOOR_INTLK,
	PE_FRNT_DOOR_INTLK,
	PE_FRNT_DOOR_OPN_REQ,
	PE_THRD_FEED_DOOR_INTLK,
	PE_FRNT_THRD_EXIT_DOOR_INTLK,
	PE_RR_FEED_DOOR_INTLK,
	PE_RR_EXIT_DOOR_INTLK,
	PE_RR_EXIT_DOOR_OPN_REQ,
	PWS_FRNT_FEED_DOOR_INTLK,
	PWS_FRNT_FEED_DOOR_OPN_REQ,
	PWS_FRNT_EXIT_DOOR_INTLK,
	PWS_RR_EXIT_DOOR_INTLK,
	PWS_RR_EXIT_DOOR_OPN_REQ,
	UIC_THRD_FEED_DOOR_INTLK,
	UIC_THRD_EXIT_DOOR_INTLK,
	EFS_1_INTRLK,
	EFS_2_INTRLK,
	PE_FRNT_EMS,
	PE_RR_EMS,
	PWS_FRNT_EMS,
	PWS_RR_EMS,
	UIC_FRNT_FEED_EMS,
	UIC_FRNT_EXIT_EMS,
	UIC_RR_EMS,
	UIC_OPER_EMS,
	UW_EMS,
	RW_EMS
)DINT;
END_TYPE

// ---- POUs/Lib/Events/Enums/eStationNo_1.TcDUT
{attribute 'qualified_only'}
//{attribute 'strict'}
{attribute 'to_string'}
TYPE eStationNo_1 :
(
	Station1 := 1,
	Station2 := 2,
	Station3 := 3,
	Station4 := 4,
	Station5 := 5,
	Station6 := 6,
	Station7 := 7
)DINT;
END_TYPE

// ---- POUs/Lib/Events/Enums/eSubsystemID_1.TcDUT
{attribute 'qualified_only'}
//{attribute 'strict'}
{attribute 'to_string'}
TYPE eSubsystemID_1 :
(
	NoSubsystem := 0,
	General ,
	Safety ,
	Blanket ,
	Station_1 ,
	Station_2 ,
	Station_3 ,
	Station_4 ,
	Station_5 ,
	Station_6 ,
	WHS ,
	ILP	,
	ImagingOil ,
	AmbientControl ,
	ELC ,
	ITM	,
	BKT_Tension	,
	BKT_Centering ,
	BR_St_1	,
	BR_St_2	,
	BR_St_3 ,
	BR_St_4	,
	BR_St_5	,
	BR_St_6	,
	BKT_Drying,
	BKT_HeatElement_1 ,
	BKT_HeatElement_2 ,
	BKT_HeatElement_3 ,
	BKT_HeatElement_4 ,
	BKT_HeatElement_5 ,
	BKT_HeatElement_6 ,
	BKT_HeatElement_7 ,
	BKT_HeatElement_8 ,
	BKT_HeatElement_9 ,
	BKT_HeatElement_10 ,
	BRU	,
	Asid_Stn_1 ,
	Asid_Stn_2 ,
	Asid_Stn_3 ,
	Asid_Stn_4 ,
	Asid_Stn_5 ,
	Asid_Stn_6 ,
	LPH_Stn_1 ,
	LPH_Stn_2 ,
	LPH_Stn_3 ,
	LPH_Stn_4 ,
	LPH_Stn_5 ,
	LPH_Stn_6 ,
	LPH_Cooling ,
	CS_Stn_1 ,
	CS_Stn_2 ,
	CS_Stn_3,
	CS_Stn_4 ,
	CS_Stn_5 ,
	CS_Stn_6 ,
	BID_Manager_1_Stn_1 ,
	BID_Manager_2_Stn_1 ,
	BID_Manager_1_Stn_2 ,
	BID_Manager_2_Stn_2 ,
	BID_Manager_1_Stn_3 ,
	BID_Manager_2_Stn_3 ,
	BID_Manager_1_Stn_4 ,
	BID_Manager_2_Stn_4 ,
	BID_Manager_1_Stn_5 ,
	BID_Manager_2_Stn_5 ,
	BID_Manager_1_Stn_6 ,
	BID_Manager_2_Stn_6 ,
	BID_Rot_1_Stn_1 ,
	BID_Rot_2_Stn_1	,
	BID_Rot_1_Stn_2	,
	BID_Rot_2_Stn_2	,
	BID_Rot_1_Stn_3	,
	BID_Rot_2_Stn_3	,
	BID_Rot_1_Stn_4	,
	BID_Rot_2_Stn_4 ,
	BID_Rot_1_Stn_5	,
	BID_Rot_2_Stn_5	,
	BID_Rot_1_Stn_6	,
	BID_Rot_2_Stn_6	,
	BID_Eng_1_Stn_1	,
	BID_Eng_2_Stn_1	,
	BID_Eng_1_Stn_2	,
	BID_Eng_2_Stn_2	,
	BID_Eng_1_Stn_3	,
	BID_Eng_2_Stn_3	,
	BID_Eng_1_Stn_4	,
	BID_Eng_2_Stn_4 ,
	BID_Eng_1_Stn_5	,
	BID_Eng_2_Stn_5	,
	BID_Eng_1_Stn_6	,
	BID_Eng_2_Stn_6	,
	BID_HV_1_Stn_1 ,
	BID_HV_2_Stn_1 ,
	BID_HV_1_Stn_2 ,
	BID_HV_2_Stn_2 ,
	BID_HV_1_Stn_3 ,
	BID_HV_2_Stn_3 ,
	BID_HV_1_Stn_4 ,
	BID_HV_2_Stn_4 ,
	BID_HV_1_Stn_5 ,
	BID_HV_2_Stn_5 ,
	BID_HV_1_Stn_6 ,
	BID_HV_2_Stn_6 ,
	INK_1_Stn_1	,
	INK_2_Stn_1	,
	INK_1_Stn_2	,
	INK_2_Stn_2 ,
	INK_1_Stn_3	,
	INK_2_Stn_3	,
	INK_1_Stn_4	,
	INK_2_Stn_4	,
	INK_1_Stn_5	,
	INK_2_Stn_5	,
	INK_1_Stn_6	,
	INK_2_Stn_6	,
	AsidChargeHV_Stn_1 ,
	AsidChargeHV_Stn_2 ,
	AsidChargeHV_Stn_3 ,
	AsidChargeHV_Stn_4 ,
	AsidChargeHV_Stn_5 ,
	AsidChargeHV_Stn_6 ,
	CR_Engage_Stn_1 ,
	CR_Engage_Stn_2 ,
	CR_Engage_Stn_3 ,
	CR_Engage_Stn_4 ,
	CR_Engage_Stn_5 ,
	CR_Engage_Stn_6 ,
	InkWater_1 ,
	InkWater_2 ,
	UW ,
	WHS_Internal ,
	WHS_Impression ,
	WHS_Buffer ,
	SPM ,
	RW ,
	Primer ,
	Dryer ,
	Corona ,
	IMO_Reservoir ,
	IMO_Recycle ,
	IMO_Waste ,
	IMO_Temperature ,
	IMO_Flow ,
	IMO_Dirtiness ,
	ITC ,
	CWS ,
	CVC ,
	Manager,
	LAST 
)DINT;
END_TYPE

// ---- POUs/Lib/Events/Enums/eVendorNameID_1.TcDUT
{attribute 'qualified_only'}
//{attribute 'strict'}
{attribute 'to_string'}
TYPE eVendorNameID_1 :
(	
	NoVendor := 		0,
	BR := 				1,
	Beckhoff := 		2,
	Elmo := 			3,
	ControlTechnique :=	4,
	Servotronics := 	5,
	Nidec :=			6,
	LAST		
)DINT;
END_TYPE

// ---- POUs/Lib/Events/Struct/EventHeader_Typ.TcDUT
TYPE EventHeader_Typ :
STRUCT
	SubsysID:		eSubsystemID;
	pFlowID:		POINTER TO DINT;	
END_STRUCT
END_TYPE

// ---- POUs/Lib/Events/Struct/EventParam_Typ.TcDUT
TYPE EventParam_Typ :
STRUCT
	MotorID:eMotorID;
	SensorID:eSensorID;
	VendorNameID:eVendorNameID;
	VendorErrorCode:DINT;
	IntParam1:DINT;
	IntParam2:DINT;
	RealParam1:REAL;	
	RealParam2:REAL;
	StringParam:STRING[64];
END_STRUCT
END_TYPE

// ---- POUs/Lib/Events/Struct/EventReport_Typ.TcDUT
TYPE EventReport_Typ :
STRUCT
	EventID:STRING;
	SubsysID:eSubsystemID;
	FlowID:DINT;
	SequentialID:DINT;
	EventType:STRING;
	MotorID:eMotorID;
	SensorID:eSensorID;
	VendorNameID:eVendorNameID;
	VendorErrorCode:DINT;
	IntParam1:DINT;
	IntParam2:DINT;
	RealParam1:REAL;	
	RealParam2:REAL;
	StringParam:STRING[64];	
END_STRUCT
END_TYPE

// ---- POUs/Lib/Inveter_Lib/Enum_INV_Ctrl.TcDUT
{attribute 'qualified_only'}
//{attribute 'strict'}
TYPE Enum_INV_Ctrl :
(
	ENV_Disable := 0,
	ENV_Run :=4,
	ENV_GetReady := 6,
	ENV_Switch_on := 7,
	ENV_Enable_operation := 15,
	ENV_Trip := 100,
	ENV_Reset_Error := 128
);
END_TYPE

// ---- POUs/Lib/Inveter_Lib/Enum_INV_Status.TcDUT
{attribute 'qualified_only'}
//{attribute 'strict'}
TYPE Enum_INV_Status :
(
	ENV_Trip := 24,
	ENV_ReadyTo_switchon :=561,
	ENV_SwitchedOn:=563,
	ENV_Operation_Enabled:=567,
	ENV_Off := 624
	
);
END_TYPE

// ---- POUs/Lib/Logging/logLib/DUTs/enumLogMessageLevelSeverity.TcDUT
//{attribute 'qualified_only'}
//{attribute 'strict'}
TYPE enumLogMessageLevelSeverity :
(
	LOG_RESERVED := 0,
	LOG_FATAL,
	LOG_ERROR,
	LOG_WARNING,
	LOG_INFO,
	LOG_DEBUG
);
END_TYPE

// ---- POUs/Lib/Logging/logLib/DUTs/E_LogStatusReport_Type.TcDUT
{attribute 'qualified_only'}
{attribute 'strict'}
TYPE E_LogStatusReport_Type :
(
	General:=	0,
	Speed,
	Eng,
	EFS

);
END_TYPE

// ---- POUs/Lib/Logging/logLib/DUTs/FailureReportMsgStruct.TcDUT
TYPE FailureReportMsgStruct :
STRUCT
	FailureType : USINT;
	FailureSubType : USINT;
	FailedUnitID : USINT;
	Severity : USINT;
	ErrorCode : UINT;
	SheetID : DINT;
	ReferenceID : UDINT;
	ActualValue : UINT;
	ViolatedThreshold : UINT;
END_STRUCT
END_TYPE

// ---- POUs/Lib/Logging/logLib/DUTs/LogArrayHandlePointers.TcDUT
TYPE LogArrayHandlePointers :
STRUCT
	writePointer : UINT := 0;
	readPointer : UINT := 0;
	numOfMembers : UINT := 0;
	isBusy : BOOL := FALSE; (*If writing to array is busy now*)
END_STRUCT
END_TYPE

// ---- POUs/Lib/Logging/logLib/DUTs/LogArrayStruct.TcDUT
TYPE LogArrayStruct :
STRUCT
	TIME_TC : TIMESTRUCT; //Oren modification to Beckhoff
	Angle : UINT;
	data : LogMsgLogData;	
END_STRUCT
END_TYPE

// ---- POUs/Lib/Logging/logLib/DUTs/LogGlobalArrayObj.TcDUT
TYPE LogGlobalArrayObj :
STRUCT
		ARRAY_TC : ARRAY[0..GLOBAL_ARRAY_LENGTH] OF LogArrayStruct; //Oren Edit array name and size
		pointers : LogArrayHandlePointers;
		SemData : LogGlobalArraySemStruct;	
		
END_STRUCT
END_TYPE

// ---- POUs/Lib/Logging/logLib/DUTs/LogGlobalArraySemStruct.TcDUT
TYPE LogGlobalArraySemStruct :
STRUCT
	//SemID : UDINT;
	//SemCreate_0 : SemCreate;
	//SemGetInfo_0 : SemGetInfo;
	SemaStat : UINT;
END_STRUCT
END_TYPE

// ---- POUs/Lib/Logging/logLib/DUTs/LogLocalArrayObj.TcDUT
TYPE LogLocalArrayObj :
STRUCT
		array_tc : ARRAY[0..LOCAL_ARRAY_LENGTH] OF LogArrayStruct;
		pointers : LogArrayHandlePointers;	
END_STRUCT
END_TYPE

// ---- POUs/Lib/Logging/logLib/DUTs/LogMsgLogData.TcDUT
TYPE LogMsgLogData :
STRUCT
		category : STRING(LOG_MSG_CATEGORY_LENGTH);
		levelSeverity : enumLogMessageLevelSeverity;
		text : STRING[LOG_MSG_TEXT_LENGTH];
		params_tc : ARRAY[0..MAX_COUNT_LOG_PARAM] OF DINT;
		noParams : BOOL;
END_STRUCT
END_TYPE

// ---- POUs/Lib/Logging/logLib/DUTs/OperationTypeEnum.TcDUT
//{attribute 'qualified_only'}
//{attribute 'strict'}
TYPE OperationTypeEnum :
(
		COLLECT2LOCAL, (*Collect a message into local array*)
		COPY2GLOBAL (*Copy messages from local array to global array*)
);
END_TYPE

// ---- POUs/Lib/Logging/PLC_ClientComm/UDP_Comm/PcComm/UDPClientHandler_typ.TcDUT
TYPE UDPClientHandler_typ :
STRUCT
		status : UDPClientOutputStatus_typ;
		no_data_received_count : UINT; (*Counts up if no data are received*)
		Udp_GetLocalAmsNetId: FB_GetLocalAmsNetId;
		UdpOpen_0 : FB_SocketUdpCreate; (*TS6310 | TwinCAT PLC Lib: TCP/IP*)
		UdpSend_0 : FB_SocketUdpSendTo; (*TS6310 | TwinCAT PLC Lib: TCP/IP*)
		SocketCloseAll_0 : FB_SocketCloseAll; (*TS6310 | TwinCAT PLC Lib: TCP/IP*)
		seq_number : UINT;
		clientId : UINT;
		InitOnCyclic : BOOL := FALSE;	
END_STRUCT
END_TYPE

// ---- POUs/Lib/Logging/PLC_ClientComm/UDP_Comm/PcComm/UDPClientOutputStatus_typ.TcDUT
TYPE UDPClientOutputStatus_typ :
STRUCT
		opened : BOOL;	
END_STRUCT
END_TYPE

// ---- POUs/Lib/Motion/CanOpenAxis/CoEDrive_Ctrl_Adr_typ.TcDUT
TYPE CoEDrive_Ctrl_Adr_typ :
STRUCT
	//output
	ControlWord      : CoE_Obj_typ;
	HomingMethod     : CoE_Obj_typ;
	HomingSWSpeed    : CoE_Obj_typ;//switch speed
	HomingTrSpeed    : CoE_Obj_typ;//Trigger spedd
	HomingAcc        : CoE_Obj_typ;
	HomeOffset       : CoE_Obj_typ;
	OperationMode    : CoE_Obj_typ;
	//Velocty Ctrl KV
	KpSpeed    		: CoE_Obj_typ;
	KISpeed    		: CoE_Obj_typ;
	GainScheduler   : CoE_Obj_typ;
	AccClosePosErr  : CoE_Obj_typ;
	//
	TorqueOffset : CoE_Obj_typ;
	MaxTorque    : CoE_Obj_typ;
	RatedCurrent     : CoE_Obj_typ;
	MaxCurrent    	 : CoE_Obj_typ;
	PositionErrorWin : CoE_Obj_typ; // Position error Window
	//input
	StatusWord       : CoE_Obj_typ;
	DCVoltage        : CoE_Obj_typ;
	
	
	
	ParamsVersionObj : CoE_Obj_typ;
	FWVersionObj     : CoE_Obj_typ;
	
END_STRUCT
END_TYPE

// ---- POUs/Lib/Motion/CanOpenAxis/CoE_FOE_Ctrl_typ.TcDUT
TYPE CoE_FOE_Ctrl_typ :
STRUCT
	Version_From_Drive:       UDINT; 
	fbEcFoeLoad_0:				FB_EcFoeLoad;
 
	fbFileOpen:					FB_FileOpen;
	fbFileClose:				FB_FileClose;	
	Foe_File_Path:				T_MaxString;
	
	hFile: 						UINT;            
END_STRUCT
END_TYPE

// ---- POUs/Lib/Motion/CanOpenAxis/DriveParID/eDS402DriveParID.TcDUT
{attribute 'qualified_only'}
{attribute 'strict'}
TYPE eDS402DriveParID :
(
	ModeOfOperation 	:= 16#6060 ,
	MotorRatedCurrent 	:= 16#6075 ,
	MotorRatedTorque 	:= 16#6076 ,
	Spare := 1
);
END_TYPE

// ---- POUs/Lib/Motion/CanOpenAxis/DriveParID/eElmoDriveParID.TcDUT
{attribute 'qualified_only'}
{attribute 'strict'}
TYPE eElmoDriveParID :
(
	RatedCurrent	:= 16#6075,
	RatedTorque		:= 16#6076,
	PCTRL_Kv := 16#6060 ,
	SCTRL_Kv := 16#6061 ,
	SCTRL_Tn := 16#6062 ,		
	Spare := 10
);
END_TYPE

// ---- POUs/Lib/Motion/CanOpenAxis/DriveParID/eNidecDriveParID.TcDUT
{attribute 'qualified_only'}
{attribute 'strict'}
TYPE eNidecDriveParID :
(
	Menue03 	:= 16#2003 ,		
	Menue04 	:= 16#2004 ,	
	Menue05 	:= 16#2005 ,
	Menue39 	:= 16#2027 ,
	PCTRL_Kv := 16#6060 ,
	SCTRL_Kv := 16#6061 ,
	SCTRL_Tn := 16#6062 ,		
	Spare := 10
);
END_TYPE

// ---- POUs/Lib/Motion/CanOpenAxis/eCaOpDriveModeOfOperation.TcDUT
{attribute 'qualified_only'}
{attribute 'strict'}
TYPE eCaOpDriveModeOfOperation :
(
	ProfilePositionMode				:= 1,
	VelocityCtrMode    				:= 2,
	ProfileVelocityMode 	   	    := 3,
	TorqueVelocityMode 				:= 4,
	HomingMode				    	:= 6,
	InterpolationPosMode			:= 7,
	CyclicSyncMode					:= 8
	
);
END_TYPE

// ---- POUs/Lib/Motion/CanOpenAxis/EcCoeSdo/EcCoeSdo_Ctrl_typ.TcDUT
TYPE EcCoeSdo_Ctrl_typ :
	STRUCT
		Input	: EcCoeSdo_Input_typ ;
		Output	: EcCoeSdo_Output_typ ;
	END_STRUCT
END_TYPE

// ---- POUs/Lib/Motion/CanOpenAxis/EcCoeSdo/EcCoeSdo_Input_typ.TcDUT
TYPE EcCoeSdo_Input_typ :
	STRUCT
		Read	: EcCoeSdo_Par_Read_typ;
		Write	: EcCoeSdo_Par_Write_typ;
	END_STRUCT
END_TYPE

// ---- POUs/Lib/Motion/CanOpenAxis/EcCoeSdo/EcCoeSdo_Output_typ.TcDUT
TYPE EcCoeSdo_Output_typ :
	STRUCT
		Read		: EcCoeSdo_Status_typ ;
		Write		: EcCoeSdo_Status_typ ;
	END_STRUCT
END_TYPE

// ---- POUs/Lib/Motion/CanOpenAxis/EcCoeSdo/EcCoeSdo_Par_Read_typ.TcDUT
TYPE EcCoeSdo_Par_Read_typ : 	
	STRUCT  (*parameter structure*)
		
        nSubIndex       : BYTE; 
        nIndex          : WORD;
		pDstBuf         : POINTER TO DWORD; 
		cbBufLen        : UDINT; 
		tTimeout        : TIME := DEFAULT_ADS_TIMEOUT; 

	END_STRUCT
END_TYPE

